LIN {X 0,Y 191.599,Z 487.439,A -85,B 0,C 180,E1 -22378.178,E2 -22378.178} C_VEL
LIN {X 0,Y 188.775,Z 497.388,A -85,B 0,C 180,E1 -22380.443,E2 -22380.443} C_VEL
LIN {X 0,Y 185.751,Z 506.671,A -85,B 0,C 180,E1 -22382.998,E2 -22382.998} C_VEL
LIN {X 0,Y 182.834,Z 515.984,A -85,B 0,C 180,E1 -22386.196,E2 -22386.196} C_VEL
LIN {X 0,Y 180.386,Z 523.716,A -85,B 0,C 180,E1 -22389.473,E2 -22389.473} C_VEL
LIN {X 0,Y 178.668,Z 530.164,A -85,B 0,C 180,E1 -22392.842,E2 -22392.842} C_VEL
LIN {X 0,Y 177.27,Z 535.423,A -85,B 0,C 180,E1 -22396.239,E2 -22396.239} C_VEL
LIN {X 0,Y 176.509,Z 539.701,A -85,B 0,C 180,E1 -22399.678,E2 -22399.678} C_VEL
LIN {X 0,Y 176.094,Z 543.09,A -85,B 0,C 180,E1 -22403.123,E2 -22403.123} C_VEL
LIN {X 0,Y 175.98,Z 546.233,A -85,B 0,C 180,E1 -22407.711,E2 -22407.711} C_VEL
LIN {X 0,Y 176.11,Z 547.274,A -85,B 0,C 180,E1 -22410,E2 -22410} C_VEL
LIN {X 0,Y 175.951,Z 548.313,A -85,B 0,C 180,E1 -22414.582,E2 -22414.582} C_VEL
LIN {X 0,Y 176.358,Z 548.034,A -85,B 0,C 180,E1 -22419.172,E2 -22419.172} C_VEL
LIN {X 0,Y 177.547,Z 546.453,A -85,B 0,C 180,E1 -22423.739,E2 -22423.739} C_VEL
LIN {X 0,Y 179.835,Z 543.544,A -85,B 0,C 180,E1 -22428.218,E2 -22428.218} C_VEL
LIN {X 0,Y 182.971,Z 539.228,A -85,B 0,C 180,E1 -22432.587,E2 -22432.587} C_VEL
LIN {X 0,Y 187.233,Z 533.386,A -85,B 0,C 180,E1 -22436.771,E2 -22436.771} C_VEL
LIN {X 0,Y 191.773,Z 526.85,A -85,B 0,C 180,E1 -22440.258,E2 -22440.258} C_VEL
LIN {X 0,Y 197.063,Z 518.782,A -85,B 0,C 180,E1 -22443.557,E2 -22443.557} C_VEL
LIN {X 0,Y 202.154,Z 510.365,A -85,B 0,C 180,E1 -22446.228,E2 -22446.228} C_VEL
LIN {X 0,Y 207.47,Z 500.385,A -85,B 0,C 180,E1 -22448.764,E2 -22448.764} C_VEL
LIN {X 0,Y 212.439,Z 490.125,A -85,B 0,C 180,E1 -22450.795,E2 -22450.795} C_VEL
LIN {X 0,Y 217.646,Z 477.789,A -85,B 0,C 180,E1 -22452.695,E2 -22452.695} C_VEL
LIN {X 0,Y 221.984,Z 465.612,A -85,B 0,C 180,E1 -22454.147,E2 -22454.147} C_VEL
LIN {X 0,Y 225.952,Z 452.09,A -85,B 0,C 180,E1 -22455.356,E2 -22455.356} C_VEL
LIN {X 0,Y 229.131,Z 437.931,A -85,B 0,C 180,E1 -22456.278,E2 -22456.278} C_VEL
LIN {X 0,Y 231.408,Z 423.369,A -85,B 0,C 180,E1 -22456.916,E2 -22456.916} C_VEL
LIN {X 0,Y 235.491,Z 369.623,A -85,B 0,C 180,E1 -22458.417,E2 -22458.417} C_VEL
LIN {X 0,Y 230.901,Z 358.639,A -85,B 0,C 180,E1 -22460.636,E2 -22460.636} C_VEL
LIN {X 0,Y 226.425,Z 349.412,A -85,B 0,C 180,E1 -22462.945,E2 -22462.945} C_VEL
LIN {X 0,Y 221.453,Z 340.153,A -85,B 0,C 180,E1 -22465.762,E2 -22465.762} C_VEL
LIN {X 0,Y 217.127,Z 332.644,A -85,B 0,C 180,E1 -22468.519,E2 -22468.519} C_VEL
LIN {X 0,Y 213.375,Z 326.679,A -85,B 0,C 180,E1 -22471.251,E2 -22471.251} C_VEL
LIN {X 0,Y 210.205,Z 321.75,A -85,B 0,C 180,E1 -22473.925,E2 -22473.925} C_VEL
LIN {X 0,Y 206.082,Z 315.639,A -85,B 0,C 180,E1 -22478.162,E2 -22478.162} C_VEL
LIN {X 0,Y 203.31,Z 313.098,A -85,B 0,C 180,E1 -22481.708,E2 -22481.708} C_VEL
LIN {X 0,Y 202.069,Z 310.201,A -85,B 0,C 180,E1 -22484.169,E2 -22484.169} C_VEL
LIN {X 0,Y 199.716,Z 308.658,A -85,B 0,C 180,E1 -22491.906,E2 -22491.906} C_VEL
LIN {X 0,Y 200.848,Z 309.272,A -85,B 0,C 180,E1 -22499.496,E2 -22499.496} C_VEL
LIN {X 0,Y 202.332,Z 310.353,A -85,B 0,C 180,E1 -22502.735,E2 -22502.735} C_VEL
LIN {X 0,Y 203.891,Z 313.395,A -85,B 0,C 180,E1 -22505.526,E2 -22505.526} C_VEL
LIN {X 0,Y 206.375,Z 315.736,A -85,B 0,C 180,E1 -22508.566,E2 -22508.566} C_VEL
LIN {X 0,Y 208.594,Z 319.275,A -85,B 0,C 180,E1 -22510.97,E2 -22510.97} C_VEL
LIN {X 0,Y 210.431,Z 321.211,A -85,B 0,C 180,E1 -22512.619,E2 -22512.619} C_VEL
LIN {X 0,Y 213.321,Z 325.119,A -85,B 0,C 180,E1 -22515.004,E2 -22515.004} C_VEL
LIN {X 0,Y 217.334,Z 330.84,A -85,B 0,C 180,E1 -22517.888,E2 -22517.888} C_VEL
LIN {X 0,Y 221.168,Z 336.313,A -85,B 0,C 180,E1 -22520.267,E2 -22520.267} C_VEL
LIN {X 0,Y 226.928,Z 345.152,A -85,B 0,C 180,E1 -22523.433,E2 -22523.433} C_VEL
LIN {X 0,Y 230.977,Z 352.505,A -85,B 0,C 180,E1 -22525.475,E2 -22525.475} C_VEL
LIN {X 0,Y 235.865,Z 362.778,A -85,B 0,C 180,E1 -22527.784,E2 -22527.784} C_VEL
LIN {X 0,Y 231.891,Z 415.14,A -85,B 0,C 180,E1 -22529.244,E2 -22529.244} C_VEL
LIN {X 0,Y 229.732,Z 429.687,A -85,B 0,C 180,E1 -22529.912,E2 -22529.912} C_VEL
LIN {X 0,Y 226.709,Z 443.815,A -85,B 0,C 180,E1 -22530.875,E2 -22530.875} C_VEL
LIN {X 0,Y 223.245,Z 456.349,A -85,B 0,C 180,E1 -22532.041,E2 -22532.041} C_VEL
LIN {X 0,Y 219.149,Z 468.478,A -85,B 0,C 180,E1 -22533.511,E2 -22533.511} C_VEL
LIN {X 0,Y 214.377,Z 480.398,A -85,B 0,C 180,E1 -22535.367,E2 -22535.367} C_VEL
LIN {X 0,Y 209.445,Z 490.898,A -85,B 0,C 180,E1 -22537.427,E2 -22537.427} C_VEL
LIN {X 0,Y 204.004,Z 501.09,A -85,B 0,C 180,E1 -22539.96,E2 -22539.96} C_VEL
LIN {X 0,Y 198.765,Z 509.97,A -85,B 0,C 180,E1 -22542.805,E2 -22542.805} C_VEL
LIN {X 0,Y 193.954,Z 517.278,A -85,B 0,C 180,E1 -22545.772,E2 -22545.772} C_VEL
LIN {X 0,Y 189.097,Z 524.169,A -85,B 0,C 180,E1 -22549.429,E2 -22549.429} C_VEL
LIN {X 0,Y 185.565,Z 528.877,A -85,B 0,C 180,E1 -22552.702,E2 -22552.702} C_VEL
LIN {X 0,Y 182.542,Z 532.562,A -85,B 0,C 180,E1 -22556.066,E2 -22556.066} C_VEL
LIN {X 0,Y 180.148,Z 535.354,A -85,B 0,C 180,E1 -22559.526,E2 -22559.526} C_VEL
LIN {X 0,Y 177.802,Z 537.718,A -85,B 0,C 180,E1 -22564.228,E2 -22564.228} C_VEL
LIN {X 0,Y 176.335,Z 538.64,A -85,B 0,C 180,E1 -22568.98,E2 -22568.98} C_VEL
LIN {X 0,Y 175.773,Z 538.153,A -85,B 0,C 180,E1 -22573.747,E2 -22573.747} C_VEL
LIN {X 0,Y 175.656,Z 536.288,A -85,B 0,C 180,E1 -22578.461,E2 -22578.461} C_VEL
LIN {X 0,Y 176.209,Z 533.006,A -85,B 0,C 180,E1 -22583.128,E2 -22583.128} C_VEL
LIN {X 0,Y 176.982,Z 529.54,A -85,B 0,C 180,E1 -22586.585,E2 -22586.585} C_VEL
LIN {X 0,Y 178.416,Z 523.586,A -85,B 0,C 180,E1 -22591.129,E2 -22591.129} C_VEL
LIN {X 0,Y 180.399,Z 516.872,A -85,B 0,C 180,E1 -22595.029,E2 -22595.029} C_VEL
LIN {X 0,Y 183.06,Z 508.512,A -85,B 0,C 180,E1 -22598.834,E2 -22598.834} C_VEL
LIN {X 0,Y 185.895,Z 499.796,A -85,B 0,C 180,E1 -22602.001,E2 -22602.001} C_VEL
LIN {X 0,Y 189.223,Z 489.232,A -85,B 0,C 180,E1 -22605.069,E2 -22605.069} C_VEL
LIN {X 0,Y 192.63,Z 477.416,A -85,B 0,C 180,E1 -22607.792,E2 -22607.792} C_VEL
LIN {X 0,Y 195.58,Z 465.587,A -85,B 0,C 180,E1 -22609.96,E2 -22609.96} C_VEL
LIN {X 0,Y 198.157,Z 454.251,A -85,B 0,C 180,E1 -22611.59,E2 -22611.59} C_VEL
LIN {X 0,Y 200.663,Z 441.026,A -85,B 0,C 180,E1 -22613.068,E2 -22613.068} C_VEL
LIN {X 0,Y 202.616,Z 426.751,A -85,B 0,C 180,E1 -22614.256,E2 -22614.256} C_VEL
LIN {X 0,Y 204.006,Z 412.463,A -85,B 0,C 180,E1 -22615.027,E2 -22615.027} C_VEL
LIN {X 0,Y 208.114,Z 340.341,A -85,B 0,C 180,E1 -22617.315,E2 -22617.315} C_VEL
LIN {X 0,Y 203.57,Z 328.395,A -85,B 0,C 180,E1 -22618.771,E2 -22618.771} C_VEL
LIN {X 0,Y 195.628,Z 313.308,A -85,B 0,C 180,E1 -22621.27,E2 -22621.27} C_VEL
LIN {X 0,Y 188.469,Z 301.599,A -85,B 0,C 180,E1 -22623.689,E2 -22623.689} C_VEL
LIN {X 0,Y 183.578,Z 294.334,A -85,B 0,C 180,E1 -22625.471,E2 -22625.471} C_VEL
LIN {X 0,Y 181.208,Z 290.635,A -85,B 0,C 180,E1 -22626.393,E2 -22626.393} C_VEL
LIN {X 0,Y 179.254,Z 288.283,A -85,B 0,C 180,E1 -22627.143,E2 -22627.143} C_VEL
LIN {X 0,Y 178.516,Z 285.874,A -85,B 0,C 180,E1 -22627.554,E2 -22627.554} C_VEL
LIN {X 0,Y 178.498,Z 285.866,A -85,B 0,C 180,E1 -22632.015,E2 -22632.015} C_VEL
LIN {X 0,Y 178.52,Z 285.859,A -85,B 0,C 180,E1 -22635.122,E2 -22635.122} C_VEL
LIN {X 0,Y 178.508,Z 285.86,A -85,B 0,C 180,E1 -22638.42,E2 -22638.42} C_VEL
LIN {X 0,Y 178.46,Z 285.851,A -85,B 0,C 180,E1 -22643.796,E2 -22643.796} C_VEL
LIN {X 0,Y 178.484,Z 285.864,A -85,B 0,C 180,E1 -22646.55,E2 -22646.55} C_VEL
LIN {X 0,Y 178.516,Z 285.865,A -85,B 0,C 180,E1 -22650.009,E2 -22650.009} C_VEL
LIN {X 0,Y 178.518,Z 285.851,A -85,B 0,C 180,E1 -22654.885,E2 -22654.885} C_VEL
LIN {X 0,Y 178.618,Z 285.853,A -85,B 0,C 180,E1 -22660.787,E2 -22660.787} C_VEL
LIN {X 0,Y 178.653,Z 285.849,A -85,B 0,C 180,E1 -22666.351,E2 -22666.351} C_VEL
LIN {X 0,Y 178.907,Z 285.804,A -85,B 0,C 180,E1 -22670.963,E2 -22670.963} C_VEL
LIN {X 0,Y 179.149,Z 285.793,A -85,B 0,C 180,E1 -22677.755,E2 -22677.755} C_VEL
LIN {X 0,Y 179.367,Z 285.757,A -85,B 0,C 180,E1 -22680.003,E2 -22680.003} C_VEL
LIN {X 0,Y 178.862,Z 285.804,A -85,B 0,C 180,E1 -22684.51,E2 -22684.51} C_VEL
LIN {X 0,Y 178.91,Z 285.821,A -85,B 0,C 180,E1 -22689.043,E2 -22689.043} C_VEL
LIN {X 0,Y 178.655,Z 285.83,A -85,B 0,C 180,E1 -22693.655,E2 -22693.655} C_VEL
LIN {X 0,Y 178.621,Z 285.852,A -85,B 0,C 180,E1 -22699.216,E2 -22699.216} C_VEL
LIN {X 0,Y 178.521,Z 285.872,A -85,B 0,C 180,E1 -22705.117,E2 -22705.117} C_VEL
LIN {X 0,Y 178.525,Z 285.871,A -85,B 0,C 180,E1 -22709.996,E2 -22709.996} C_VEL
LIN {X 0,Y 178.487,Z 285.873,A -85,B 0,C 180,E1 -22714.221,E2 -22714.221} C_VEL
LIN {X 0,Y 178.461,Z 286.066,A -85,B 0,C 180,E1 -22718.1,E2 -22718.1} C_VEL
LIN {X 0,Y 179.328,Z 288.615,A -85,B 0,C 180,E1 -22718.527,E2 -22718.527} C_VEL
LIN {X 0,Y 181.633,Z 291.388,A -85,B 0,C 180,E1 -22719.409,E2 -22719.409} C_VEL
LIN {X 0,Y 184,Z 294.886,A -85,B 0,C 180,E1 -22720.314,E2 -22720.314} C_VEL
LIN {X 0,Y 187.709,Z 300.898,A -85,B 0,C 180,E1 -22721.688,E2 -22721.688} C_VEL
LIN {X 0,Y 194.217,Z 313.493,A -85,B 0,C 180,E1 -22724.019,E2 -22724.019} C_VEL
LIN {X 0,Y 200.32,Z 326.993,A -85,B 0,C 180,E1 -22726.083,E2 -22726.083} C_VEL
LIN {X 0,Y 206.79,Z 344.301,A -85,B 0,C 180,E1 -22728.211,E2 -22728.211} C_VEL
LIN {X 0,Y 207.653,Z 350.597,A -85,B 0,C 180,E1 -22728.65,E2 -22728.65} C_VEL
LIN {X 0,Y 205.055,Z 399.727,A -85,B 0,C 180,E1 -22730.218,E2 -22730.218} C_VEL
LIN {X 0,Y 204.232,Z 405.578,A -85,B 0,C 180,E1 -22730.296,E2 -22730.296} C_VEL
LIN {X 0,Y 198.314,Z 424.511,A -85,B 0,C 180,E1 -22730.052,E2 -22730.052} C_VEL
LIN {X 0,Y 197.12,Z 430.265,A -85,B 0,C 180,E1 -22730.247,E2 -22730.247} C_VEL
LIN {X 0,Y 195.345,Z 443.358,A -85,B 0,C 180,E1 -22731.146,E2 -22731.146} C_VEL
LIN {X 0,Y 192.903,Z 456.479,A -85,B 0,C 180,E1 -22732.393,E2 -22732.393} C_VEL
LIN {X 0,Y 189.9,Z 469.458,A -85,B 0,C 180,E1 -22734.044,E2 -22734.044} C_VEL
LIN {X 0,Y 186.72,Z 482.513,A -85,B 0,C 180,E1 -22736.278,E2 -22736.278} C_VEL
LIN {X 0,Y 183.793,Z 492.107,A -85,B 0,C 180,E1 -22738.28,E2 -22738.28} C_VEL
LIN {X 0,Y 180.587,Z 502.213,A -85,B 0,C 180,E1 -22740.892,E2 -22740.892} C_VEL
LIN {X 0,Y 177.225,Z 512.26,A -85,B 0,C 180,E1 -22744.138,E2 -22744.138} C_VEL
LIN {X 0,Y 174.538,Z 520.595,A -85,B 0,C 180,E1 -22747.511,E2 -22747.511} C_VEL
LIN {X 0,Y 172.095,Z 528.543,A -85,B 0,C 180,E1 -22751.549,E2 -22751.549} C_VEL
LIN {X 0,Y 170.328,Z 534.902,A -85,B 0,C 180,E1 -22755.666,E2 -22755.666} C_VEL
LIN {X 0,Y 169.291,Z 540.513,A -85,B 0,C 180,E1 -22760.441,E2 -22760.441} C_VEL
LIN {X 0,Y 169.015,Z 542.701,A -85,B 0,C 180,E1 -22762.834,E2 -22762.834} C_VEL
LIN {X 0,Y 168.894,Z 545.923,A -85,B 0,C 180,E1 -22767.615,E2 -22767.615} C_VEL
LIN {X 0,Y 169.017,Z 546.996,A -85,B 0,C 180,E1 -22770,E2 -22770} C_VEL
LIN {X 0,Y 168.865,Z 548.097,A -85,B 0,C 180,E1 -22774.774,E2 -22774.774} C_VEL
LIN {X 0,Y 169.328,Z 547.881,A -85,B 0,C 180,E1 -22779.556,E2 -22779.556} C_VEL
LIN {X 0,Y 170.609,Z 546.362,A -85,B 0,C 180,E1 -22784.309,E2 -22784.309} C_VEL
LIN {X 0,Y 173.061,Z 543.518,A -85,B 0,C 180,E1 -22788.958,E2 -22788.958} C_VEL
LIN {X 0,Y 176.655,Z 538.932,A -85,B 0,C 180,E1 -22793.785,E2 -22793.785} C_VEL
LIN {X 0,Y 180.898,Z 533.512,A -85,B 0,C 180,E1 -22797.787,E2 -22797.787} C_VEL
LIN {X 0,Y 185.656,Z 527.059,A -85,B 0,C 180,E1 -22801.365,E2 -22801.365} C_VEL
LIN {X 0,Y 191.196,Z 519.083,A -85,B 0,C 180,E1 -22804.732,E2 -22804.732} C_VEL
LIN {X 0,Y 196.487,Z 510.766,A -85,B 0,C 180,E1 -22807.448,E2 -22807.448} C_VEL
LIN {X 0,Y 202.357,Z 500.267,A -85,B 0,C 180,E1 -22810.172,E2 -22810.172} C_VEL
LIN {X 0,Y 207.688,Z 489.714,A -85,B 0,C 180,E1 -22812.263,E2 -22812.263} C_VEL
LIN {X 0,Y 213.051,Z 477.329,A -85,B 0,C 180,E1 -22814.174,E2 -22814.174} C_VEL
LIN {X 0,Y 217.574,Z 465.082,A -85,B 0,C 180,E1 -22815.615,E2 -22815.615} C_VEL
LIN {X 0,Y 221.628,Z 451.483,A -85,B 0,C 180,E1 -22816.83,E2 -22816.83} C_VEL
LIN {X 0,Y 224.944,Z 437.181,A -85,B 0,C 180,E1 -22817.736,E2 -22817.736} C_VEL
LIN {X 0,Y 227.194,Z 423.145,A -85,B 0,C 180,E1 -22818.339,E2 -22818.339} C_VEL
LIN {X 0,Y 231.149,Z 372.075,A -85,B 0,C 180,E1 -22819.801,E2 -22819.801} C_VEL
LIN {X 0,Y 226.57,Z 361.295,A -85,B 0,C 180,E1 -22822.17,E2 -22822.17} C_VEL
LIN {X 0,Y 222.235,Z 352.184,A -85,B 0,C 180,E1 -22824.597,E2 -22824.597} C_VEL
LIN {X 0,Y 217.151,Z 342.693,A -85,B 0,C 180,E1 -22827.752,E2 -22827.752} C_VEL
LIN {X 0,Y 212.407,Z 334.425,A -85,B 0,C 180,E1 -22831.201,E2 -22831.201} C_VEL
LIN {X 0,Y 208.423,Z 328.16,A -85,B 0,C 180,E1 -22834.648,E2 -22834.648} C_VEL
LIN {X 0,Y 204.763,Z 322.459,A -85,B 0,C 180,E1 -22838.61,E2 -22838.61} C_VEL
LIN {X 0,Y 202.118,Z 319.903,A -85,B 0,C 180,E1 -22842.17,E2 -22842.17} C_VEL
LIN {X 0,Y 200.885,Z 317.174,A -85,B 0,C 180,E1 -22844.729,E2 -22844.729} C_VEL
LIN {X 0,Y 198.844,Z 315.713,A -85,B 0,C 180,E1 -22851.87,E2 -22851.87} C_VEL
LIN {X 0,Y 199.968,Z 316.325,A -85,B 0,C 180,E1 -22859.494,E2 -22859.494} C_VEL
LIN {X 0,Y 201.222,Z 317.276,A -85,B 0,C 180,E1 -22862.327,E2 -22862.327} C_VEL
LIN {X 0,Y 202.8,Z 320.36,A -85,B 0,C 180,E1 -22865.263,E2 -22865.263} C_VEL
LIN {X 0,Y 205.027,Z 322.627,A -85,B 0,C 180,E1 -22868.113,E2 -22868.113} C_VEL
LIN {X 0,Y 207.417,Z 326.287,A -85,B 0,C 180,E1 -22870.755,E2 -22870.755} C_VEL
LIN {X 0,Y 208.836,Z 327.902,A -85,B 0,C 180,E1 -22872.077,E2 -22872.077} C_VEL
LIN {X 0,Y 212.21,Z 332.715,A -85,B 0,C 180,E1 -22874.946,E2 -22874.946} C_VEL
LIN {X 0,Y 215.576,Z 337.605,A -85,B 0,C 180,E1 -22877.426,E2 -22877.426} C_VEL
LIN {X 0,Y 220.029,Z 344.131,A -85,B 0,C 180,E1 -22880.249,E2 -22880.249} C_VEL
LIN {X 0,Y 225.73,Z 353.527,A -85,B 0,C 180,E1 -22883.442,E2 -22883.442} C_VEL
LIN {X 0,Y 230.588,Z 363.521,A -85,B 0,C 180,E1 -22885.947,E2 -22885.947} C_VEL
LIN {X 0,Y 231.586,Z 365.841,A -85,B 0,C 180,E1 -22886.443,E2 -22886.443} C_VEL
LIN {X 0,Y 227.745,Z 414.733,A -85,B 0,C 180,E1 -22887.804,E2 -22887.804} C_VEL
LIN {X 0,Y 225.513,Z 429.496,A -85,B 0,C 180,E1 -22888.471,E2 -22888.471} C_VEL
LIN {X 0,Y 222.393,Z 443.676,A -85,B 0,C 180,E1 -22889.425,E2 -22889.425} C_VEL
LIN {X 0,Y 218.866,Z 456.059,A -85,B 0,C 180,E1 -22890.563,E2 -22890.563} C_VEL
LIN {X 0,Y 214.572,Z 468.45,A -85,B 0,C 180,E1 -22892.062,E2 -22892.062} C_VEL
LIN {X 0,Y 209.611,Z 480.408,A -85,B 0,C 180,E1 -22893.92,E2 -22893.92} C_VEL
LIN {X 0,Y 203.966,Z 491.947,A -85,B 0,C 180,E1 -22896.209,E2 -22896.209} C_VEL
LIN {X 0,Y 198.318,Z 501.969,A -85,B 0,C 180,E1 -22898.775,E2 -22898.775} C_VEL
LIN {X 0,Y 192.874,Z 510.714,A -85,B 0,C 180,E1 -22901.672,E2 -22901.672} C_VEL
LIN {X 0,Y 187.85,Z 517.932,A -85,B 0,C 180,E1 -22904.698,E2 -22904.698} C_VEL
LIN {X 0,Y 183.465,Z 523.866,A -85,B 0,C 180,E1 -22907.906,E2 -22907.906} C_VEL
LIN {X 0,Y 179.213,Z 529.174,A -85,B 0,C 180,E1 -22911.652,E2 -22911.652} C_VEL
LIN {X 0,Y 175.409,Z 533.532,A -85,B 0,C 180,E1 -22915.881,E2 -22915.881} C_VEL
LIN {X 0,Y 172.262,Z 536.754,A -85,B 0,C 180,E1 -22920.688,E2 -22920.688} C_VEL
LIN {X 0,Y 170.184,Z 538.489,A -85,B 0,C 180,E1 -22925.61,E2 -22925.61} C_VEL
LIN {X 0,Y 168.945,Z 538.803,A -85,B 0,C 180,E1 -22930.562,E2 -22930.562} C_VEL
LIN {X 0,Y 168.674,Z 538.361,A -85,B 0,C 180,E1 -22933.387,E2 -22933.387} C_VEL
LIN {X 0,Y 168.53,Z 536.661,A -85,B 0,C 180,E1 -22937.966,E2 -22937.966} C_VEL
LIN {X 0,Y 169.046,Z 533.488,A -85,B 0,C 180,E1 -22942.836,E2 -22942.836} C_VEL
LIN {X 0,Y 169.829,Z 530.109,A -85,B 0,C 180,E1 -22946.441,E2 -22946.441} C_VEL
LIN {X 0,Y 171.302,Z 524.262,A -85,B 0,C 180,E1 -22951.176,E2 -22951.176} C_VEL
LIN {X 0,Y 173.302,Z 517.678,A -85,B 0,C 180,E1 -22955.235,E2 -22955.235} C_VEL
LIN {X 0,Y 176.021,Z 509.508,A -85,B 0,C 180,E1 -22959.19,E2 -22959.19} C_VEL
LIN {X 0,Y 178.96,Z 500.948,A -85,B 0,C 180,E1 -22962.474,E2 -22962.474} C_VEL
LIN {X 0,Y 182.367,Z 490.582,A -85,B 0,C 180,E1 -22965.65,E2 -22965.65} C_VEL
LIN {X 0,Y 185.915,Z 478.99,A -85,B 0,C 180,E1 -22968.457,E2 -22968.457} C_VEL
LIN {X 0,Y 188.984,Z 467.448,A -85,B 0,C 180,E1 -22970.688,E2 -22970.688} C_VEL
LIN {X 0,Y 191.538,Z 456.54,A -85,B 0,C 180,E1 -22972.376,E2 -22972.376} C_VEL
LIN {X 0,Y 194.173,Z 443.872,A -85,B 0,C 180,E1 -22973.886,E2 -22973.886} C_VEL
LIN {X 0,Y 196.319,Z 429.762,A -85,B 0,C 180,E1 -22975.157,E2 -22975.157} C_VEL
LIN {X 0,Y 197.909,Z 415.615,A -85,B 0,C 180,E1 -22976.013,E2 -22976.013} C_VEL
LIN {X 0,Y 199.359,Z 392.322,A -85,B 0,C 180,E1 -22976.843,E2 -22976.843} C_VEL
LIN {X 0,Y 202.207,Z 341.799,A -85,B 0,C 180,E1 -22978.472,E2 -22978.472} C_VEL
LIN {X 0,Y 198.36,Z 331.838,A -85,B 0,C 180,E1 -22979.766,E2 -22979.766} C_VEL
LIN {X 0,Y 191.132,Z 317.879,A -85,B 0,C 180,E1 -22982.17,E2 -22982.17} C_VEL
LIN {X 0,Y 184.087,Z 306.206,A -85,B 0,C 180,E1 -22984.686,E2 -22984.686} C_VEL
LIN {X 0,Y 178.777,Z 298.299,A -85,B 0,C 180,E1 -22986.731,E2 -22986.731} C_VEL
LIN {X 0,Y 177.03,Z 295.69,A -85,B 0,C 180,E1 -22987.446,E2 -22987.446} C_VEL
LIN {X 0,Y 174.901,Z 292.466,A -85,B 0,C 180,E1 -22988.353,E2 -22988.353} C_VEL
LIN {X 0,Y 174.113,Z 291.47,A -85,B 0,C 180,E1 -22988.686,E2 -22988.686} C_VEL
LIN {X 0,Y 172.088,Z 289.03,A -85,B 0,C 180,E1 -22989.559,E2 -22989.559} C_VEL
LIN {X 0,Y 171.411,Z 286.741,A -85,B 0,C 180,E1 -22990.023,E2 -22990.023} C_VEL
LIN {X 0,Y 171.442,Z 286.751,A -85,B 0,C 180,E1 -22994.177,E2 -22994.177} C_VEL
LIN {X 0,Y 171.425,Z 286.748,A -85,B 0,C 180,E1 -22999.012,E2 -22999.012} C_VEL
LIN {X 0,Y 171.434,Z 286.74,A -85,B 0,C 180,E1 -23002.058,E2 -23002.058} C_VEL
LIN {X 0,Y 171.421,Z 286.754,A -85,B 0,C 180,E1 -23007.797,E2 -23007.797} C_VEL
LIN {X 0,Y 171.442,Z 286.739,A -85,B 0,C 180,E1 -23010.537,E2 -23010.537} C_VEL
LIN {X 0,Y 171.447,Z 286.74,A -85,B 0,C 180,E1 -23015.804,E2 -23015.804} C_VEL
LIN {X 0,Y 171.574,Z 286.73,A -85,B 0,C 180,E1 -23020.875,E2 -23020.875} C_VEL
LIN {X 0,Y 171.571,Z 286.729,A -85,B 0,C 180,E1 -23025.776,E2 -23025.776} C_VEL
LIN {X 0,Y 171.844,Z 286.687,A -85,B 0,C 180,E1 -23030.588,E2 -23030.588} C_VEL
LIN {X 0,Y 171.811,Z 286.688,A -85,B 0,C 180,E1 -23035.311,E2 -23035.311} C_VEL
LIN {X 0,Y 172.329,Z 286.633,A -85,B 0,C 180,E1 -23040.003,E2 -23040.003} C_VEL
LIN {X 0,Y 171.811,Z 286.683,A -85,B 0,C 180,E1 -23044.696,E2 -23044.696} C_VEL
LIN {X 0,Y 171.847,Z 286.697,A -85,B 0,C 180,E1 -23049.418,E2 -23049.418} C_VEL
LIN {X 0,Y 171.573,Z 286.716,A -85,B 0,C 180,E1 -23054.231,E2 -23054.231} C_VEL
LIN {X 0,Y 171.54,Z 286.734,A -85,B 0,C 180,E1 -23059.56,E2 -23059.56} C_VEL
LIN {X 0,Y 171.46,Z 286.753,A -85,B 0,C 180,E1 -23065.612,E2 -23065.612} C_VEL
LIN {X 0,Y 171.443,Z 286.75,A -85,B 0,C 180,E1 -23070.589,E2 -23070.589} C_VEL
LIN {X 0,Y 171.393,Z 286.814,A -85,B 0,C 180,E1 -23075.668,E2 -23075.668} C_VEL
LIN {X 0,Y 172.308,Z 289.471,A -85,B 0,C 180,E1 -23076.17,E2 -23076.17} C_VEL
LIN {X 0,Y 174.335,Z 291.706,A -85,B 0,C 180,E1 -23077.029,E2 -23077.029} C_VEL
LIN {X 0,Y 176.961,Z 295.713,A -85,B 0,C 180,E1 -23078.158,E2 -23078.158} C_VEL
LIN {X 0,Y 178.596,Z 298.091,A -85,B 0,C 180,E1 -23078.827,E2 -23078.827} C_VEL
LIN {X 0,Y 182.642,Z 304.082,A -85,B 0,C 180,E1 -23080.405,E2 -23080.405} C_VEL
LIN {X 0,Y 189.835,Z 318.338,A -85,B 0,C 180,E1 -23083.14,E2 -23083.14} C_VEL
LIN {X 0,Y 195.529,Z 331.21,A -85,B 0,C 180,E1 -23085.176,E2 -23085.176} C_VEL
LIN {X 0,Y 201.519,Z 347.777,A -85,B 0,C 180,E1 -23087.273,E2 -23087.273} C_VEL
LIN {X 0,Y 201.822,Z 352.981,A -85,B 0,C 180,E1 -23087.566,E2 -23087.566} C_VEL
LIN {X 0,Y 197.799,Z 423.508,A -85,B 0,C 180,E1 -23089.906,E2 -23089.906} C_VEL
LIN {X 0,Y 197.12,Z 430.265,A -85,B 0,C 180,E1 -23090.247,E2 -23090.247} C_VEL
LIN {X 0,Y 196.033,Z 434.097,A -85,B 0,C 180,E1 -23090.355,E2 -23090.355} C_VEL
LIN {X 0,Y 189.413,Z 445.895,A -85,B 0,C 180,E1 -23090.283,E2 -23090.283} C_VEL
LIN {X 0,Y 188.223,Z 449.593,A -85,B 0,C 180,E1 -23090.533,E2 -23090.533} C_VEL
LIN {X 0,Y 185.525,Z 462.569,A -85,B 0,C 180,E1 -23092.007,E2 -23092.007} C_VEL
LIN {X 0,Y 182.835,Z 473.325,A -85,B 0,C 180,E1 -23093.568,E2 -23093.568} C_VEL
LIN {X 0,Y 179.691,Z 485.184,A -85,B 0,C 180,E1 -23095.79,E2 -23095.79} C_VEL
LIN {X 0,Y 177.365,Z 492.134,A -85,B 0,C 180,E1 -23097.325,E2 -23097.325} C_VEL
LIN {X 0,Y 174.359,Z 501.302,A -85,B 0,C 180,E1 -23099.746,E2 -23099.746} C_VEL
LIN {X 0,Y 170.81,Z 511.469,A -85,B 0,C 180,E1 -23103.09,E2 -23103.09} C_VEL
LIN {X 0,Y 167.941,Z 519.902,A -85,B 0,C 180,E1 -23106.575,E2 -23106.575} C_VEL
LIN {X 0,Y 165.681,Z 526.92,A -85,B 0,C 180,E1 -23110.163,E2 -23110.163} C_VEL
LIN {X 0,Y 163.914,Z 532.727,A -85,B 0,C 180,E1 -23113.818,E2 -23113.818} C_VEL
LIN {X 0,Y 162.699,Z 537.434,A -85,B 0,C 180,E1 -23117.527,E2 -23117.527} C_VEL
LIN {X 0,Y 162.105,Z 541.219,A -85,B 0,C 180,E1 -23121.272,E2 -23121.272} C_VEL
LIN {X 0,Y 161.801,Z 544.136,A -85,B 0,C 180,E1 -23125.016,E2 -23125.016} C_VEL
LIN {X 0,Y 161.927,Z 546.716,A -85,B 0,C 180,E1 -23130,E2 -23130} C_VEL
LIN {X 0,Y 161.804,Z 547.466,A -85,B 0,C 180,E1 -23132.489,E2 -23132.489} C_VEL
LIN {X 0,Y 161.937,Z 547.967,A -85,B 0,C 180,E1 -23137.481,E2 -23137.481} C_VEL
LIN {X 0,Y 162.876,Z 547.163,A -85,B 0,C 180,E1 -23142.459,E2 -23142.459} C_VEL
LIN {X 0,Y 164.878,Z 545.055,A -85,B 0,C 180,E1 -23147.36,E2 -23147.36} C_VEL
LIN {X 0,Y 167.986,Z 541.594,A -85,B 0,C 180,E1 -23152.118,E2 -23152.118} C_VEL
LIN {X 0,Y 172.103,Z 536.682,A -85,B 0,C 180,E1 -23156.691,E2 -23156.691} C_VEL
LIN {X 0,Y 177.403,Z 530.176,A -85,B 0,C 180,E1 -23160.997,E2 -23160.997} C_VEL
LIN {X 0,Y 182.803,Z 522.975,A -85,B 0,C 180,E1 -23164.545,E2 -23164.545} C_VEL
LIN {X 0,Y 189.043,Z 514.105,A -85,B 0,C 180,E1 -23167.836,E2 -23167.836} C_VEL
LIN {X 0,Y 194.748,Z 504.847,A -85,B 0,C 180,E1 -23170.508,E2 -23170.508} C_VEL
LIN {X 0,Y 200.333,Z 494.655,A -85,B 0,C 180,E1 -23172.819,E2 -23172.819} C_VEL
LIN {X 0,Y 205.854,Z 483.44,A -85,B 0,C 180,E1 -23174.759,E2 -23174.759} C_VEL
LIN {X 0,Y 210.929,Z 471.105,A -85,B 0,C 180,E1 -23176.442,E2 -23176.442} C_VEL
LIN {X 0,Y 215.136,Z 459.206,A -85,B 0,C 180,E1 -23177.654,E2 -23177.654} C_VEL
LIN {X 0,Y 218.765,Z 446.242,A -85,B 0,C 180,E1 -23178.67,E2 -23178.67} C_VEL
LIN {X 0,Y 221.684,Z 432.344,A -85,B 0,C 180,E1 -23179.451,E2 -23179.451} C_VEL
LIN {X 0,Y 223.65,Z 417.686,A -85,B 0,C 180,E1 -23180.007,E2 -23180.007} C_VEL
LIN {X 0,Y 226.984,Z 374.911,A -85,B 0,C 180,E1 -23181.207,E2 -23181.207} C_VEL
LIN {X 0,Y 223.064,Z 365.487,A -85,B 0,C 180,E1 -23183.38,E2 -23183.38} C_VEL
LIN {X 0,Y 219.422,Z 357.561,A -85,B 0,C 180,E1 -23185.552,E2 -23185.552} C_VEL
LIN {X 0,Y 214.653,Z 348.38,A -85,B 0,C 180,E1 -23188.686,E2 -23188.686} C_VEL
LIN {X 0,Y 210.267,Z 340.346,A -85,B 0,C 180,E1 -23192.097,E2 -23192.097} C_VEL
LIN {X 0,Y 206.633,Z 334.465,A -85,B 0,C 180,E1 -23195.43,E2 -23195.43} C_VEL
LIN {X 0,Y 203.338,Z 329.247,A -85,B 0,C 180,E1 -23199.191,E2 -23199.191} C_VEL
LIN {X 0,Y 200.776,Z 326.405,A -85,B 0,C 180,E1 -23202.938,E2 -23202.938} C_VEL
LIN {X 0,Y 199.898,Z 324.18,A -85,B 0,C 180,E1 -23204.927,E2 -23204.927} C_VEL
LIN {X 0,Y 197.97,Z 322.761,A -85,B 0,C 180,E1 -23211.834,E2 -23211.834} C_VEL
LIN {X 0,Y 199.082,Z 323.383,A -85,B 0,C 180,E1 -23219.492,E2 -23219.492} C_VEL
LIN {X 0,Y 200.101,Z 324.14,A -85,B 0,C 180,E1 -23221.872,E2 -23221.872} C_VEL
LIN {X 0,Y 201.658,Z 327.257,A -85,B 0,C 180,E1 -23224.915,E2 -23224.915} C_VEL
LIN {X 0,Y 203.684,Z 329.475,A -85,B 0,C 180,E1 -23227.639,E2 -23227.639} C_VEL
LIN {X 0,Y 206.374,Z 333.468,A -85,B 0,C 180,E1 -23230.668,E2 -23230.668} C_VEL
LIN {X 0,Y 207.46,Z 334.939,A -85,B 0,C 180,E1 -23231.725,E2 -23231.725} C_VEL
LIN {X 0,Y 210.475,Z 339.308,A -85,B 0,C 180,E1 -23234.377,E2 -23234.377} C_VEL
LIN {X 0,Y 213.704,Z 344.18,A -85,B 0,C 180,E1 -23236.856,E2 -23236.856} C_VEL
LIN {X 0,Y 217.593,Z 350.062,A -85,B 0,C 180,E1 -23239.445,E2 -23239.445} C_VEL
LIN {X 0,Y 222.928,Z 359.153,A -85,B 0,C 180,E1 -23242.589,E2 -23242.589} C_VEL
LIN {X 0,Y 227.401,Z 368.697,A -85,B 0,C 180,E1 -23245.023,E2 -23245.023} C_VEL
LIN {X 0,Y 223.648,Z 415.206,A -85,B 0,C 180,E1 -23246.341,E2 -23246.341} C_VEL
LIN {X 0,Y 221.344,Z 429.92,A -85,B 0,C 180,E1 -23247.009,E2 -23247.009} C_VEL
LIN {X 0,Y 218.219,Z 443.605,A -85,B 0,C 180,E1 -23247.916,E2 -23247.916} C_VEL
LIN {X 0,Y 214.472,Z 456.382,A -85,B 0,C 180,E1 -23249.088,E2 -23249.088} C_VEL
LIN {X 0,Y 210.131,Z 468.471,A -85,B 0,C 180,E1 -23250.548,E2 -23250.548} C_VEL
LIN {X 0,Y 204.997,Z 480.451,A -85,B 0,C 180,E1 -23252.413,E2 -23252.413} C_VEL
LIN {X 0,Y 199.325,Z 491.639,A -85,B 0,C 180,E1 -23254.63,E2 -23254.63} C_VEL
LIN {X 0,Y 193.757,Z 501.229,A -85,B 0,C 180,E1 -23257.064,E2 -23257.064} C_VEL
LIN {X 0,Y 187.959,Z 510.154,A -85,B 0,C 180,E1 -23259.96,E2 -23259.96} C_VEL
LIN {X 0,Y 182.679,Z 517.498,A -85,B 0,C 180,E1 -23263.034,E2 -23263.034} C_VEL
LIN {X 0,Y 177.952,Z 523.523,A -85,B 0,C 180,E1 -23266.281,E2 -23266.281} C_VEL
LIN {X 0,Y 172.878,Z 529.521,A -85,B 0,C 180,E1 -23270.564,E2 -23270.564} C_VEL
LIN {X 0,Y 169.236,Z 533.421,A -85,B 0,C 180,E1 -23274.453,E2 -23274.453} C_VEL
LIN {X 0,Y 165.788,Z 536.791,A -85,B 0,C 180,E1 -23279.424,E2 -23279.424} C_VEL
LIN {X 0,Y 163.406,Z 538.632,A -85,B 0,C 180,E1 -23284.572,E2 -23284.572} C_VEL
LIN {X 0,Y 161.977,Z 539.035,A -85,B 0,C 180,E1 -23289.69,E2 -23289.69} C_VEL
LIN {X 0,Y 161.631,Z 538.558,A -85,B 0,C 180,E1 -23293.043,E2 -23293.043} C_VEL
LIN {X 0,Y 161.419,Z 537.035,A -85,B 0,C 180,E1 -23297.427,E2 -23297.427} C_VEL
LIN {X 0,Y 161.888,Z 533.958,A -85,B 0,C 180,E1 -23302.517,E2 -23302.517} C_VEL
LIN {X 0,Y 162.679,Z 530.678,A -85,B 0,C 180,E1 -23306.285,E2 -23306.285} C_VEL
LIN {X 0,Y 164.19,Z 524.938,A -85,B 0,C 180,E1 -23311.227,E2 -23311.227} C_VEL
LIN {X 0,Y 166.184,Z 518.475,A -85,B 0,C 180,E1 -23315.46,E2 -23315.46} C_VEL
LIN {X 0,Y 169.004,Z 510.443,A -85,B 0,C 180,E1 -23319.575,E2 -23319.575} C_VEL
LIN {X 0,Y 172.018,Z 502.033,A -85,B 0,C 180,E1 -23322.986,E2 -23322.986} C_VEL
LIN {X 0,Y 175.545,Z 491.904,A -85,B 0,C 180,E1 -23326.275,E2 -23326.275} C_VEL
LIN {X 0,Y 179.23,Z 480.549,A -85,B 0,C 180,E1 -23329.172,E2 -23329.172} C_VEL
LIN {X 0,Y 182.428,Z 469.285,A -85,B 0,C 180,E1 -23331.468,E2 -23331.468} C_VEL
LIN {X 0,Y 184.972,Z 458.774,A -85,B 0,C 180,E1 -23333.216,E2 -23333.216} C_VEL
LIN {X 0,Y 187.77,Z 446.619,A -85,B 0,C 180,E1 -23334.754,E2 -23334.754} C_VEL
LIN {X 0,Y 190.066,Z 432.694,A -85,B 0,C 180,E1 -23336.12,E2 -23336.12} C_VEL
LIN {X 0,Y 191.822,Z 418.327,A -85,B 0,C 180,E1 -23337.081,E2 -23337.081} C_VEL
LIN {X 0,Y 193.142,Z 399.928,A -85,B 0,C 180,E1 -23337.809,E2 -23337.809} C_VEL
LIN {X 0,Y 196.442,Z 343.511,A -85,B 0,C 180,E1 -23339.667,E2 -23339.667} C_VEL
LIN {X 0,Y 193.301,Z 335.429,A -85,B 0,C 180,E1 -23340.783,E2 -23340.783} C_VEL
LIN {X 0,Y 186.27,Z 321.653,A -85,B 0,C 180,E1 -23343.267,E2 -23343.267} C_VEL
LIN {X 0,Y 178.708,Z 309.051,A -85,B 0,C 180,E1 -23346.149,E2 -23346.149} C_VEL
LIN {X 0,Y 172.941,Z 300.564,A -85,B 0,C 180,E1 -23348.55,E2 -23348.55} C_VEL
LIN {X 0,Y 170.39,Z 296.894,A -85,B 0,C 180,E1 -23349.696,E2 -23349.696} C_VEL
LIN {X 0,Y 168.139,Z 293.746,A -85,B 0,C 180,E1 -23350.752,E2 -23350.752} C_VEL
LIN {X 0,Y 167.402,Z 292.599,A -85,B 0,C 180,E1 -23351.117,E2 -23351.117} C_VEL
LIN {X 0,Y 165.4,Z 290.497,A -85,B 0,C 180,E1 -23352.069,E2 -23352.069} C_VEL
LIN {X 0,Y 164.389,Z 287.63,A -85,B 0,C 180,E1 -23352.696,E2 -23352.696} C_VEL
LIN {X 0,Y 164.386,Z 287.608,A -85,B 0,C 180,E1 -23356.845,E2 -23356.845} C_VEL
LIN {X 0,Y 164.369,Z 287.633,A -85,B 0,C 180,E1 -23360.32,E2 -23360.32} C_VEL
LIN {X 0,Y 164.34,Z 287.606,A -85,B 0,C 180,E1 -23364.343,E2 -23364.343} C_VEL
LIN {X 0,Y 164.398,Z 287.628,A -85,B 0,C 180,E1 -23369.141,E2 -23369.141} C_VEL
LIN {X 0,Y 164.404,Z 287.603,A -85,B 0,C 180,E1 -23374.696,E2 -23374.696} C_VEL
LIN {X 0,Y 164.479,Z 287.614,A -85,B 0,C 180,E1 -23380.054,E2 -23380.054} C_VEL
LIN {X 0,Y 164.501,Z 287.61,A -85,B 0,C 180,E1 -23385.151,E2 -23385.151} C_VEL
LIN {X 0,Y 164.764,Z 287.572,A -85,B 0,C 180,E1 -23390.18,E2 -23390.18} C_VEL
LIN {X 0,Y 164.827,Z 287.541,A -85,B 0,C 180,E1 -23392.654,E2 -23392.654} C_VEL
LIN {X 0,Y 165.044,Z 287.55,A -85,B 0,C 180,E1 -23397.563,E2 -23397.563} C_VEL
LIN {X 0,Y 165.292,Z 287.509,A -85,B 0,C 180,E1 -23400.003,E2 -23400.003} C_VEL
LIN {X 0,Y 164.759,Z 287.562,A -85,B 0,C 180,E1 -23404.897,E2 -23404.897} C_VEL
LIN {X 0,Y 164.829,Z 287.578,A -85,B 0,C 180,E1 -23407.352,E2 -23407.352} C_VEL
LIN {X 0,Y 164.702,Z 287.567,A -85,B 0,C 180,E1 -23411.064,E2 -23411.064} C_VEL
LIN {X 0,Y 164.482,Z 287.622,A -85,B 0,C 180,E1 -23417.406,E2 -23417.406} C_VEL
LIN {X 0,Y 164.474,Z 287.616,A -85,B 0,C 180,E1 -23419.992,E2 -23419.992} C_VEL
LIN {X 0,Y 164.388,Z 287.632,A -85,B 0,C 180,E1 -23426.131,E2 -23426.131} C_VEL
LIN {X 0,Y 164.381,Z 287.633,A -85,B 0,C 180,E1 -23432.377,E2 -23432.377} C_VEL
LIN {X 0,Y 164.337,Z 287.641,A -85,B 0,C 180,E1 -23432.906,E2 -23432.906} C_VEL
LIN {X 0,Y 165.25,Z 290.365,A -85,B 0,C 180,E1 -23433.481,E2 -23433.481} C_VEL
LIN {X 0,Y 167.246,Z 292.53,A -85,B 0,C 180,E1 -23434.436,E2 -23434.436} C_VEL
LIN {X 0,Y 167.907,Z 293.297,A -85,B 0,C 180,E1 -23434.747,E2 -23434.747} C_VEL
LIN {X 0,Y 170.099,Z 296.641,A -85,B 0,C 180,E1 -23435.799,E2 -23435.799} C_VEL
LIN {X 0,Y 171.406,Z 298.414,A -85,B 0,C 180,E1 -23436.391,E2 -23436.391} C_VEL
LIN {X 0,Y 176.879,Z 306.338,A -85,B 0,C 180,E1 -23438.741,E2 -23438.741} C_VEL
LIN {X 0,Y 180.372,Z 312.545,A -85,B 0,C 180,E1 -23440.183,E2 -23440.183} C_VEL
LIN {X 0,Y 186.76,Z 325.894,A -85,B 0,C 180,E1 -23442.704,E2 -23442.704} C_VEL
LIN {X 0,Y 192.113,Z 339.01,A -85,B 0,C 180,E1 -23444.725,E2 -23444.725} C_VEL
LIN {X 0,Y 196.031,Z 350.366,A -85,B 0,C 180,E1 -23446.182,E2 -23446.182} C_VEL
LIN {X 0,Y 196.047,Z 355.298,A -85,B 0,C 180,E1 -23446.412,E2 -23446.412} C_VEL
LIN {X 0,Y 192.065,Z 422.729,A -85,B 0,C 180,E1 -23448.686,E2 -23448.686} C_VEL
LIN {X 0,Y 190.422,Z 437.008,A -85,B 0,C 180,E1 -23449.509,E2 -23449.509} C_VEL
LIN {X 0,Y 188.223,Z 449.593,A -85,B 0,C 180,E1 -23450.533,E2 -23450.533} C_VEL
LIN {X 0,Y 187.276,Z 453.306,A -85,B 0,C 180,E1 -23450.87,E2 -23450.87} C_VEL
LIN {X 0,Y 184.105,Z 460.43,A -85,B 0,C 180,E1 -23451.365,E2 -23451.365} C_VEL
LIN {X 0,Y 177.514,Z 472.256,A -85,B 0,C 180,E1 -23452.356,E2 -23452.356} C_VEL
LIN {X 0,Y 175.627,Z 477.217,A -85,B 0,C 180,E1 -23453.122,E2 -23453.122} C_VEL
LIN {X 0,Y 172.924,Z 486.512,A -85,B 0,C 180,E1 -23455.003,E2 -23455.003} C_VEL
LIN {X 0,Y 170.325,Z 494.319,A -85,B 0,C 180,E1 -23456.858,E2 -23456.858} C_VEL
LIN {X 0,Y 166.844,Z 503.981,A -85,B 0,C 180,E1 -23459.637,E2 -23459.637} C_VEL
LIN {X 0,Y 163.326,Z 513.678,A -85,B 0,C 180,E1 -23463.14,E2 -23463.14} C_VEL
LIN {X 0,Y 160.221,Z 522.345,A -85,B 0,C 180,E1 -23467.102,E2 -23467.102} C_VEL
LIN {X 0,Y 158.212,Z 528.355,A -85,B 0,C 180,E1 -23470.539,E2 -23470.539} C_VEL
LIN {X 0,Y 156.504,Z 533.854,A -85,B 0,C 180,E1 -23474.369,E2 -23474.369} C_VEL
LIN {X 0,Y 155.207,Z 539.615,A -85,B 0,C 180,E1 -23479.565,E2 -23479.565} C_VEL
LIN {X 0,Y 154.908,Z 541.881,A -85,B 0,C 180,E1 -23482.177,E2 -23482.177} C_VEL
LIN {X 0,Y 154.705,Z 545.267,A -85,B 0,C 180,E1 -23487.396,E2 -23487.396} C_VEL
LIN {X 0,Y 154.827,Z 546.418,A -85,B 0,C 180,E1 -23490,E2 -23490} C_VEL
LIN {X 0,Y 154.696,Z 547.657,A -85,B 0,C 180,E1 -23495.213,E2 -23495.213} C_VEL
LIN {X 0,Y 155.286,Z 547.573,A -85,B 0,C 180,E1 -23500.429,E2 -23500.429} C_VEL
LIN {X 0,Y 156.799,Z 546.187,A -85,B 0,C 180,E1 -23505.6,E2 -23505.6} C_VEL
LIN {X 0,Y 159.596,Z 543.48,A -85,B 0,C 180,E1 -23510.627,E2 -23510.627} C_VEL
LIN {X 0,Y 163.398,Z 539.38,A -85,B 0,C 180,E1 -23515.474,E2 -23515.474} C_VEL
LIN {X 0,Y 168.417,Z 533.767,A -85,B 0,C 180,E1 -23520.049,E2 -23520.049} C_VEL
LIN {X 0,Y 174.518,Z 526.474,A -85,B 0,C 180,E1 -23524.317,E2 -23524.317} C_VEL
LIN {X 0,Y 179.699,Z 519.694,A -85,B 0,C 180,E1 -23527.314,E2 -23527.314} C_VEL
LIN {X 0,Y 185.455,Z 511.592,A -85,B 0,C 180,E1 -23530.107,E2 -23530.107} C_VEL
LIN {X 0,Y 191.28,Z 502.173,A -85,B 0,C 180,E1 -23532.703,E2 -23532.703} C_VEL
LIN {X 0,Y 196.901,Z 492.181,A -85,B 0,C 180,E1 -23534.823,E2 -23534.823} C_VEL
LIN {X 0,Y 202.651,Z 480.498,A -85,B 0,C 180,E1 -23536.741,E2 -23536.741} C_VEL
LIN {X 0,Y 207.348,Z 469.112,A -85,B 0,C 180,E1 -23538.216,E2 -23538.216} C_VEL
LIN {X 0,Y 211.708,Z 456.752,A -85,B 0,C 180,E1 -23539.407,E2 -23539.407} C_VEL
LIN {X 0,Y 215.433,Z 443.112,A -85,B 0,C 180,E1 -23540.416,E2 -23540.416} C_VEL
LIN {X 0,Y 218.34,Z 428.761,A -85,B 0,C 180,E1 -23541.143,E2 -23541.143} C_VEL
LIN {X 0,Y 220.044,Z 414.846,A -85,B 0,C 180,E1 -23541.616,E2 -23541.616} C_VEL
LIN {X 0,Y 222.992,Z 377.875,A -85,B 0,C 180,E1 -23542.644,E2 -23542.644} C_VEL
LIN {X 0,Y 219.22,Z 368.572,A -85,B 0,C 180,E1 -23544.906,E2 -23544.906} C_VEL
LIN {X 0,Y 214.738,Z 358.951,A -85,B 0,C 180,E1 -23547.834,E2 -23547.834} C_VEL
LIN {X 0,Y 211.343,Z 352.334,A -85,B 0,C 180,E1 -23550.334,E2 -23550.334} C_VEL
LIN {X 0,Y 207.792,Z 345.701,A -85,B 0,C 180,E1 -23553.351,E2 -23553.351} C_VEL
LIN {X 0,Y 204.923,Z 340.855,A -85,B 0,C 180,E1 -23556.18,E2 -23556.18} C_VEL
LIN {X 0,Y 202.051,Z 336.081,A -85,B 0,C 180,E1 -23559.643,E2 -23559.643} C_VEL
LIN {X 0,Y 199.51,Z 333.003,A -85,B 0,C 180,E1 -23563.629,E2 -23563.629} C_VEL
LIN {X 0,Y 198.817,Z 331.129,A -85,B 0,C 180,E1 -23565.334,E2 -23565.334} C_VEL
LIN {X 0,Y 197.094,Z 329.817,A -85,B 0,C 180,E1 -23571.797,E2 -23571.797} C_VEL
LIN {X 0,Y 198.199,Z 330.418,A -85,B 0,C 180,E1 -23579.489,E2 -23579.489} C_VEL
LIN {X 0,Y 199.063,Z 331.239,A -85,B 0,C 180,E1 -23581.603,E2 -23581.603} C_VEL
LIN {X 0,Y 200.661,Z 334.332,A -85,B 0,C 180,E1 -23584.784,E2 -23584.784} C_VEL
LIN {X 0,Y 202.368,Z 336.333,A -85,B 0,C 180,E1 -23587.177,E2 -23587.177} C_VEL
LIN {X 0,Y 205.054,Z 340.318,A -85,B 0,C 180,E1 -23590.301,E2 -23590.301} C_VEL
LIN {X 0,Y 208.646,Z 345.727,A -85,B 0,C 180,E1 -23593.699,E2 -23593.699} C_VEL
LIN {X 0,Y 211.963,Z 350.853,A -85,B 0,C 180,E1 -23596.352,E2 -23596.352} C_VEL
LIN {X 0,Y 216.221,Z 357.805,A -85,B 0,C 180,E1 -23599.297,E2 -23599.297} C_VEL
LIN {X 0,Y 220.39,Z 365.22,A -85,B 0,C 180,E1 -23601.841,E2 -23601.841} C_VEL
LIN {X 0,Y 223.43,Z 371.851,A -85,B 0,C 180,E1 -23603.598,E2 -23603.598} C_VEL
LIN {X 0,Y 219.763,Z 415.135,A -85,B 0,C 180,E1 -23604.8,E2 -23604.8} C_VEL
LIN {X 0,Y 217.441,Z 429.708,A -85,B 0,C 180,E1 -23605.451,E2 -23605.451} C_VEL
LIN {X 0,Y 214.215,Z 443.543,A -85,B 0,C 180,E1 -23606.356,E2 -23606.356} C_VEL
LIN {X 0,Y 210.118,Z 457.021,A -85,B 0,C 180,E1 -23607.585,E2 -23607.585} C_VEL
LIN {X 0,Y 205.249,Z 469.988,A -85,B 0,C 180,E1 -23609.175,E2 -23609.175} C_VEL
LIN {X 0,Y 199.943,Z 481.732,A -85,B 0,C 180,E1 -23611.045,E2 -23611.045} C_VEL
LIN {X 0,Y 194.467,Z 492.018,A -85,B 0,C 180,E1 -23613.117,E2 -23613.117} C_VEL
LIN {X 0,Y 188.308,Z 502.161,A -85,B 0,C 180,E1 -23615.735,E2 -23615.735} C_VEL
LIN {X 0,Y 182.129,Z 511.126,A -85,B 0,C 180,E1 -23618.749,E2 -23618.749} C_VEL
LIN {X 0,Y 175.881,Z 519.221,A -85,B 0,C 180,E1 -23622.337,E2 -23622.337} C_VEL
LIN {X 0,Y 171.05,Z 524.99,A -85,B 0,C 180,E1 -23625.696,E2 -23625.696} C_VEL
LIN {X 0,Y 166.636,Z 529.847,A -85,B 0,C 180,E1 -23629.385,E2 -23629.385} C_VEL
LIN {X 0,Y 163.192,Z 533.306,A -85,B 0,C 180,E1 -23632.922,E2 -23632.922} C_VEL
LIN {X 0,Y 159.388,Z 536.792,A -85,B 0,C 180,E1 -23638.055,E2 -23638.055} C_VEL
LIN {X 0,Y 156.702,Z 538.759,A -85,B 0,C 180,E1 -23643.354,E2 -23643.354} C_VEL
LIN {X 0,Y 155.073,Z 539.265,A -85,B 0,C 180,E1 -23648.743,E2 -23648.743} C_VEL
LIN {X 0,Y 154.437,Z 538.368,A -85,B 0,C 180,E1 -23654.155,E2 -23654.155} C_VEL
LIN {X 0,Y 154.413,Z 536.091,A -85,B 0,C 180,E1 -23659.511,E2 -23659.511} C_VEL
LIN {X 0,Y 155.242,Z 532.387,A -85,B 0,C 180,E1 -23664.806,E2 -23664.806} C_VEL
LIN {X 0,Y 156.137,Z 528.63,A -85,B 0,C 180,E1 -23668.711,E2 -23668.711} C_VEL
LIN {X 0,Y 157.538,Z 523.972,A -85,B 0,C 180,E1 -23672.557,E2 -23672.557} C_VEL
LIN {X 0,Y 159.871,Z 517.193,A -85,B 0,C 180,E1 -23676.944,E2 -23676.944} C_VEL
LIN {X 0,Y 162.477,Z 510.112,A -85,B 0,C 180,E1 -23680.593,E2 -23680.593} C_VEL
LIN {X 0,Y 165.689,Z 501.592,A -85,B 0,C 180,E1 -23684.117,E2 -23684.117} C_VEL
LIN {X 0,Y 169.289,Z 491.654,A -85,B 0,C 180,E1 -23687.398,E2 -23687.398} C_VEL
LIN {X 0,Y 172.914,Z 480.921,A -85,B 0,C 180,E1 -23690.211,E2 -23690.211} C_VEL
LIN {X 0,Y 176.241,Z 469.696,A -85,B 0,C 180,E1 -23692.57,E2 -23692.57} C_VEL
LIN {X 0,Y 178.891,Z 459.217,A -85,B 0,C 180,E1 -23694.362,E2 -23694.362} C_VEL
LIN {X 0,Y 182.009,Z 446.066,A -85,B 0,C 180,E1 -23696.054,E2 -23696.054} C_VEL
LIN {X 0,Y 184.407,Z 431.831,A -85,B 0,C 180,E1 -23697.445,E2 -23697.445} C_VEL
LIN {X 0,Y 186.174,Z 417.646,A -85,B 0,C 180,E1 -23698.386,E2 -23698.386} C_VEL
LIN {X 0,Y 187.551,Z 398.199,A -85,B 0,C 180,E1 -23699.152,E2 -23699.152} C_VEL
LIN {X 0,Y 190.813,Z 345.483,A -85,B 0,C 180,E1 -23700.907,E2 -23700.907} C_VEL
LIN {X 0,Y 188.158,Z 338.72,A -85,B 0,C 180,E1 -23701.906,E2 -23701.906} C_VEL
LIN {X 0,Y 181.217,Z 325.078,A -85,B 0,C 180,E1 -23704.516,E2 -23704.516} C_VEL
LIN {X 0,Y 174.665,Z 313.956,A -85,B 0,C 180,E1 -23707.171,E2 -23707.171} C_VEL
LIN {X 0,Y 168.825,Z 305.236,A -85,B 0,C 180,E1 -23709.757,E2 -23709.757} C_VEL
LIN {X 0,Y 166.504,Z 301.953,A -85,B 0,C 180,E1 -23710.861,E2 -23710.861} C_VEL
LIN {X 0,Y 163.873,Z 298.191,A -85,B 0,C 180,E1 -23712.186,E2 -23712.186} C_VEL
LIN {X 0,Y 161.601,Z 295.183,A -85,B 0,C 180,E1 -23713.379,E2 -23713.379} C_VEL
LIN {X 0,Y 160.779,Z 293.77,A -85,B 0,C 180,E1 -23713.848,E2 -23713.848} C_VEL
LIN {X 0,Y 158.461,Z 291.637,A -85,B 0,C 180,E1 -23715.084,E2 -23715.084} C_VEL
LIN {X 0,Y 157.411,Z 289.116,A -85,B 0,C 180,E1 -23715.787,E2 -23715.787} C_VEL
LIN {X 0,Y 157.3,Z 288.492,A -85,B 0,C 180,E1 -23715.979,E2 -23715.979} C_VEL
LIN {X 0,Y 157.284,Z 288.511,A -85,B 0,C 180,E1 -23721.281,E2 -23721.281} C_VEL
LIN {X 0,Y 157.287,Z 288.484,A -85,B 0,C 180,E1 -23724.493,E2 -23724.493} C_VEL
LIN {X 0,Y 157.295,Z 288.514,A -85,B 0,C 180,E1 -23728.094,E2 -23728.094} C_VEL
LIN {X 0,Y 157.31,Z 288.477,A -85,B 0,C 180,E1 -23733.468,E2 -23733.468} C_VEL
LIN {X 0,Y 157.388,Z 288.498,A -85,B 0,C 180,E1 -23739.671,E2 -23739.671} C_VEL
LIN {X 0,Y 157.437,Z 288.492,A -85,B 0,C 180,E1 -23744.468,E2 -23744.468} C_VEL
LIN {X 0,Y 157.685,Z 288.457,A -85,B 0,C 180,E1 -23749.734,E2 -23749.734} C_VEL
LIN {X 0,Y 157.764,Z 288.42,A -85,B 0,C 180,E1 -23752.323,E2 -23752.323} C_VEL
LIN {X 0,Y 158.254,Z 288.385,A -85,B 0,C 180,E1 -23760.003,E2 -23760.003} C_VEL
LIN {X 0,Y 157.766,Z 288.458,A -85,B 0,C 180,E1 -23767.683,E2 -23767.683} C_VEL
LIN {X 0,Y 157.633,Z 288.445,A -85,B 0,C 180,E1 -23771.234,E2 -23771.234} C_VEL
LIN {X 0,Y 157.441,Z 288.49,A -85,B 0,C 180,E1 -23775.539,E2 -23775.539} C_VEL
LIN {X 0,Y 157.368,Z 288.508,A -85,B 0,C 180,E1 -23780.936,E2 -23780.936} C_VEL
LIN {X 0,Y 157.312,Z 288.51,A -85,B 0,C 180,E1 -23786.684,E2 -23786.684} C_VEL
LIN {X 0,Y 157.285,Z 288.518,A -85,B 0,C 180,E1 -23789.72,E2 -23789.72} C_VEL
LIN {X 0,Y 158.277,Z 291.294,A -85,B 0,C 180,E1 -23790.433,E2 -23790.433} C_VEL
LIN {X 0,Y 160.585,Z 293.614,A -85,B 0,C 180,E1 -23791.684,E2 -23791.684} C_VEL
LIN {X 0,Y 163.216,Z 297.585,A -85,B 0,C 180,E1 -23793.118,E2 -23793.118} C_VEL
LIN {X 0,Y 164.732,Z 299.383,A -85,B 0,C 180,E1 -23793.873,E2 -23793.873} C_VEL
LIN {X 0,Y 171.119,Z 308.651,A -85,B 0,C 180,E1 -23796.915,E2 -23796.915} C_VEL
LIN {X 0,Y 174.601,Z 314.229,A -85,B 0,C 180,E1 -23798.447,E2 -23798.447} C_VEL
LIN {X 0,Y 181.111,Z 327.7,A -85,B 0,C 180,E1 -23801.221,E2 -23801.221} C_VEL
LIN {X 0,Y 186.162,Z 339.914,A -85,B 0,C 180,E1 -23803.256,E2 -23803.256} C_VEL
LIN {X 0,Y 190.542,Z 352.608,A -85,B 0,C 180,E1 -23804.995,E2 -23804.995} C_VEL
LIN {X 0,Y 186.332,Z 422.64,A -85,B 0,C 180,E1 -23807.425,E2 -23807.425} C_VEL
LIN {X 0,Y 184.529,Z 437.372,A -85,B 0,C 180,E1 -23808.294,E2 -23808.294} C_VEL
LIN {X 0,Y 181.975,Z 451.407,A -85,B 0,C 180,E1 -23809.511,E2 -23809.511} C_VEL
LIN {X 0,Y 178.973,Z 464.472,A -85,B 0,C 180,E1 -23811.076,E2 -23811.076} C_VEL
LIN {X 0,Y 175.627,Z 477.217,A -85,B 0,C 180,E1 -23813.122,E2 -23813.122} C_VEL
LIN {X 0,Y 174.137,Z 480.554,A -85,B 0,C 180,E1 -23813.644,E2 -23813.644} C_VEL
LIN {X 0,Y 170.044,Z 485.633,A -85,B 0,C 180,E1 -23814.233,E2 -23814.233} C_VEL
LIN {X 0,Y 165.843,Z 490.606,A -85,B 0,C 180,E1 -23814.915,E2 -23814.915} C_VEL
LIN {X 0,Y 164.202,Z 493.637,A -85,B 0,C 180,E1 -23815.59,E2 -23815.59} C_VEL
LIN {X 0,Y 160.705,Z 503.048,A -85,B 0,C 180,E1 -23818.347,E2 -23818.347} C_VEL
LIN {X 0,Y 156.958,Z 512.865,A -85,B 0,C 180,E1 -23821.956,E2 -23821.956} C_VEL
LIN {X 0,Y 153.881,Z 520.99,A -85,B 0,C 180,E1 -23825.73,E2 -23825.73} C_VEL
LIN {X 0,Y 151.116,Z 528.763,A -85,B 0,C 180,E1 -23830.295,E2 -23830.295} C_VEL
LIN {X 0,Y 149.134,Z 534.959,A -85,B 0,C 180,E1 -23834.978,E2 -23834.978} C_VEL
LIN {X 0,Y 148.199,Z 539.161,A -85,B 0,C 180,E1 -23839.065,E2 -23839.065} C_VEL
LIN {X 0,Y 147.84,Z 541.462,A -85,B 0,C 180,E1 -23841.801,E2 -23841.801} C_VEL
LIN {X 0,Y 147.616,Z 544.919,A -85,B 0,C 180,E1 -23847.271,E2 -23847.271} C_VEL
LIN {X 0,Y 147.728,Z 546.104,A -85,B 0,C 180,E1 -23850,E2 -23850} C_VEL
LIN {X 0,Y 147.615,Z 546.928,A -85,B 0,C 180,E1 -23852.729,E2 -23852.729} C_VEL
LIN {X 0,Y 147.815,Z 547.57,A -85,B 0,C 180,E1 -23858.2,E2 -23858.2} C_VEL
LIN {X 0,Y 148.971,Z 546.907,A -85,B 0,C 180,E1 -23863.643,E2 -23863.643} C_VEL
LIN {X 0,Y 151.299,Z 544.943,A -85,B 0,C 180,E1 -23868.974,E2 -23868.974} C_VEL
LIN {X 0,Y 154.843,Z 541.628,A -85,B 0,C 180,E1 -23874.109,E2 -23874.109} C_VEL
LIN {X 0,Y 159.489,Z 536.869,A -85,B 0,C 180,E1 -23878.993,E2 -23878.993} C_VEL
LIN {X 0,Y 165.351,Z 530.529,A -85,B 0,C 180,E1 -23883.541,E2 -23883.541} C_VEL
LIN {X 0,Y 171.304,Z 523.511,A -85,B 0,C 180,E1 -23887.238,E2 -23887.238} C_VEL
LIN {X 0,Y 178.05,Z 514.854,A -85,B 0,C 180,E1 -23890.637,E2 -23890.637} C_VEL
LIN {X 0,Y 184.717,Z 505.114,A -85,B 0,C 180,E1 -23893.56,E2 -23893.56} C_VEL
LIN {X 0,Y 190.806,Z 494.966,A -85,B 0,C 180,E1 -23895.908,E2 -23895.908} C_VEL
LIN {X 0,Y 196.703,Z 483.926,A -85,B 0,C 180,E1 -23897.847,E2 -23897.847} C_VEL
LIN {X 0,Y 202.119,Z 471.811,A -85,B 0,C 180,E1 -23899.518,E2 -23899.518} C_VEL
LIN {X 0,Y 207.206,Z 458.229,A -85,B 0,C 180,E1 -23900.882,E2 -23900.882} C_VEL
LIN {X 0,Y 211.035,Z 445.098,A -85,B 0,C 180,E1 -23901.883,E2 -23901.883} C_VEL
LIN {X 0,Y 214.158,Z 430.835,A -85,B 0,C 180,E1 -23902.638,E2 -23902.638} C_VEL
LIN {X 0,Y 216.118,Z 416.618,A -85,B 0,C 180,E1 -23903.151,E2 -23903.151} C_VEL
LIN {X 0,Y 219.095,Z 380.75,A -85,B 0,C 180,E1 -23904.161,E2 -23904.161} C_VEL
LIN {X 0,Y 215.218,Z 371.147,A -85,B 0,C 180,E1 -23906.685,E2 -23906.685} C_VEL
LIN {X 0,Y 210.513,Z 360.865,A -85,B 0,C 180,E1 -23910.128,E2 -23910.128} C_VEL
LIN {X 0,Y 206.215,Z 352.43,A -85,B 0,C 180,E1 -23913.867,E2 -23913.867} C_VEL
LIN {X 0,Y 203.207,Z 347.149,A -85,B 0,C 180,E1 -23916.993,E2 -23916.993} C_VEL
LIN {X 0,Y 200.648,Z 342.769,A -85,B 0,C 180,E1 -23920.273,E2 -23920.273} C_VEL
LIN {X 0,Y 198.337,Z 339.733,A -85,B 0,C 180,E1 -23924.185,E2 -23924.185} C_VEL
LIN {X 0,Y 197.803,Z 338.181,A -85,B 0,C 180,E1 -23925.596,E2 -23925.596} C_VEL
LIN {X 0,Y 196.218,Z 336.873,A -85,B 0,C 180,E1 -23931.76,E2 -23931.76} C_VEL
LIN {X 0,Y 197.138,Z 337.34,A -85,B 0,C 180,E1 -23938.976,E2 -23938.976} C_VEL
LIN {X 0,Y 197.985,Z 338.131,A -85,B 0,C 180,E1 -23941.192,E2 -23941.192} C_VEL
LIN {X 0,Y 199.526,Z 341.226,A -85,B 0,C 180,E1 -23944.424,E2 -23944.424} C_VEL
LIN {X 0,Y 201.027,Z 343.074,A -85,B 0,C 180,E1 -23946.647,E2 -23946.647} C_VEL
LIN {X 0,Y 203.741,Z 347.168,A -85,B 0,C 180,E1 -23949.929,E2 -23949.929} C_VEL
LIN {X 0,Y 206.929,Z 352.246,A -85,B 0,C 180,E1 -23953.081,E2 -23953.081} C_VEL
LIN {X 0,Y 211.023,Z 358.819,A -85,B 0,C 180,E1 -23956.442,E2 -23956.442} C_VEL
LIN {X 0,Y 215.232,Z 366.185,A -85,B 0,C 180,E1 -23959.392,E2 -23959.392} C_VEL
LIN {X 0,Y 218.536,Z 372.637,A -85,B 0,C 180,E1 -23961.474,E2 -23961.474} C_VEL
LIN {X 0,Y 219.563,Z 375.04,A -85,B 0,C 180,E1 -23962.107,E2 -23962.107} C_VEL
LIN {X 0,Y 215.955,Z 415.792,A -85,B 0,C 180,E1 -23963.237,E2 -23963.237} C_VEL
LIN {X 0,Y 213.535,Z 430.35,A -85,B 0,C 180,E1 -23963.889,E2 -23963.889} C_VEL
LIN {X 0,Y 210.375,Z 443.48,A -85,B 0,C 180,E1 -23964.739,E2 -23964.739} C_VEL
LIN {X 0,Y 206.155,Z 457.01,A -85,B 0,C 180,E1 -23965.957,E2 -23965.957} C_VEL
LIN {X 0,Y 201.049,Z 470.142,A -85,B 0,C 180,E1 -23967.547,E2 -23967.547} C_VEL
LIN {X 0,Y 195.612,Z 481.793,A -85,B 0,C 180,E1 -23969.397,E2 -23969.397} C_VEL
LIN {X 0,Y 189.685,Z 492.515,A -85,B 0,C 180,E1 -23971.554,E2 -23971.554} C_VEL
LIN {X 0,Y 184.01,Z 501.426,A -85,B 0,C 180,E1 -23973.831,E2 -23973.831} C_VEL
LIN {X 0,Y 177.986,Z 510.004,A -85,B 0,C 180,E1 -23976.654,E2 -23976.654} C_VEL
LIN {X 0,Y 171.868,Z 517.748,A -85,B 0,C 180,E1 -23979.942,E2 -23979.942} C_VEL
LIN {X 0,Y 165.749,Z 524.72,A -85,B 0,C 180,E1 -23983.879,E2 -23983.879} C_VEL
LIN {X 0,Y 160.513,Z 530.154,A -85,B 0,C 180,E1 -23988.097,E2 -23988.097} C_VEL
LIN {X 0,Y 157.251,Z 533.196,A -85,B 0,C 180,E1 -23991.268,E2 -23991.268} C_VEL
LIN {X 0,Y 153.058,Z 536.781,A -85,B 0,C 180,E1 -23996.565,E2 -23996.565} C_VEL
LIN {X 0,Y 150.06,Z 538.862,A -85,B 0,C 180,E1 -24002.074,E2 -24002.074} C_VEL
LIN {X 0,Y 148.181,Z 539.495,A -85,B 0,C 180,E1 -24007.703,E2 -24007.703} C_VEL
LIN {X 0,Y 147.405,Z 538.692,A -85,B 0,C 180,E1 -24013.378,E2 -24013.378} C_VEL
LIN {X 0,Y 147.281,Z 536.508,A -85,B 0,C 180,E1 -24018.997,E2 -24018.997} C_VEL
LIN {X 0,Y 148.059,Z 532.9,A -85,B 0,C 180,E1 -24024.553,E2 -24024.553} C_VEL
LIN {X 0,Y 149,Z 529.242,A -85,B 0,C 180,E1 -24028.649,E2 -24028.649} C_VEL
LIN {X 0,Y 150.436,Z 524.646,A -85,B 0,C 180,E1 -24032.678,E2 -24032.678} C_VEL
LIN {X 0,Y 152.814,Z 518.007,A -85,B 0,C 180,E1 -24037.266,E2 -24037.266} C_VEL
LIN {X 0,Y 156.018,Z 509.745,A -85,B 0,C 180,E1 -24041.695,E2 -24041.695} C_VEL
LIN {X 0,Y 159.414,Z 501.112,A -85,B 0,C 180,E1 -24045.338,E2 -24045.338} C_VEL
LIN {X 0,Y 163.23,Z 491.036,A -85,B 0,C 180,E1 -24048.709,E2 -24048.709} C_VEL
LIN {X 0,Y 167.019,Z 480.124,A -85,B 0,C 180,E1 -24051.604,E2 -24051.604} C_VEL
LIN {X 0,Y 170.844,Z 467.286,A -85,B 0,C 180,E1 -24054.291,E2 -24054.291} C_VEL
LIN {X 0,Y 173.805,Z 456.176,A -85,B 0,C 180,E1 -24056.087,E2 -24056.087} C_VEL
LIN {X 0,Y 176.553,Z 444.359,A -85,B 0,C 180,E1 -24057.564,E2 -24057.564} C_VEL
LIN {X 0,Y 178.961,Z 430.217,A -85,B 0,C 180,E1 -24058.916,E2 -24058.916} C_VEL
LIN {X 0,Y 180.702,Z 416.26,A -85,B 0,C 180,E1 -24059.808,E2 -24059.808} C_VEL
LIN {X 0,Y 182.548,Z 389.882,A -85,B 0,C 180,E1 -24060.788,E2 -24060.788} C_VEL
LIN {X 0,Y 185.284,Z 347.472,A -85,B 0,C 180,E1 -24062.218,E2 -24062.218} C_VEL
LIN {X 0,Y 182.863,Z 341.549,A -85,B 0,C 180,E1 -24063.178,E2 -24063.178} C_VEL
LIN {X 0,Y 176.55,Z 329.02,A -85,B 0,C 180,E1 -24065.705,E2 -24065.705} C_VEL
LIN {X 0,Y 170.198,Z 318.184,A -85,B 0,C 180,E1 -24068.452,E2 -24068.452} C_VEL
LIN {X 0,Y 163.675,Z 308.138,A -85,B 0,C 180,E1 -24071.593,E2 -24071.593} C_VEL
LIN {X 0,Y 160.088,Z 303.285,A -85,B 0,C 180,E1 -24073.478,E2 -24073.478} C_VEL
LIN {X 0,Y 157.424,Z 299.519,A -85,B 0,C 180,E1 -24074.992,E2 -24074.992} C_VEL
LIN {X 0,Y 155.077,Z 296.796,A -85,B 0,C 180,E1 -24076.368,E2 -24076.368} C_VEL
LIN {X 0,Y 153.882,Z 294.7,A -85,B 0,C 180,E1 -24077.161,E2 -24077.161} C_VEL
LIN {X 0,Y 151.619,Z 292.796,A -85,B 0,C 180,E1 -24078.565,E2 -24078.565} C_VEL
LIN {X 0,Y 150.41,Z 290.301,A -85,B 0,C 180,E1 -24079.481,E2 -24079.481} C_VEL
LIN {X 0,Y 150.25,Z 289.39,A -85,B 0,C 180,E1 -24079.758,E2 -24079.758} C_VEL
LIN {X 0,Y 150.231,Z 289.369,A -85,B 0,C 180,E1 -24082.681,E2 -24082.681} C_VEL
LIN {X 0,Y 150.217,Z 289.39,A -85,B 0,C 180,E1 -24087.366,E2 -24087.366} C_VEL
LIN {X 0,Y 150.236,Z 289.357,A -85,B 0,C 180,E1 -24092.723,E2 -24092.723} C_VEL
LIN {X 0,Y 150.346,Z 289.377,A -85,B 0,C 180,E1 -24099.212,E2 -24099.212} C_VEL
LIN {X 0,Y 150.349,Z 289.38,A -85,B 0,C 180,E1 -24103.716,E2 -24103.716} C_VEL
LIN {X 0,Y 150.607,Z 289.344,A -85,B 0,C 180,E1 -24109.246,E2 -24109.246} C_VEL
LIN {X 0,Y 150.685,Z 289.302,A -85,B 0,C 180,E1 -24111.96,E2 -24111.96} C_VEL
LIN {X 0,Y 151.215,Z 289.261,A -85,B 0,C 180,E1 -24120.004,E2 -24120.004} C_VEL
LIN {X 0,Y 150.703,Z 289.339,A -85,B 0,C 180,E1 -24128.046,E2 -24128.046} C_VEL
LIN {X 0,Y 150.575,Z 289.321,A -85,B 0,C 180,E1 -24131.436,E2 -24131.436} C_VEL
LIN {X 0,Y 150.353,Z 289.379,A -85,B 0,C 180,E1 -24136.291,E2 -24136.291} C_VEL
LIN {X 0,Y 150.351,Z 289.38,A -85,B 0,C 180,E1 -24140.794,E2 -24140.794} C_VEL
LIN {X 0,Y 150.239,Z 289.395,A -85,B 0,C 180,E1 -24145.954,E2 -24145.954} C_VEL
LIN {X 0,Y 151.126,Z 292.003,A -85,B 0,C 180,E1 -24146.712,E2 -24146.712} C_VEL
LIN {X 0,Y 152.942,Z 294.158,A -85,B 0,C 180,E1 -24147.917,E2 -24147.917} C_VEL
LIN {X 0,Y 154.332,Z 295.277,A -85,B 0,C 180,E1 -24148.754,E2 -24148.754} C_VEL
LIN {X 0,Y 156.296,Z 298.382,A -85,B 0,C 180,E1 -24150.001,E2 -24150.001} C_VEL
LIN {X 0,Y 158.006,Z 300.328,A -85,B 0,C 180,E1 -24150.978,E2 -24150.978} C_VEL
LIN {X 0,Y 160.577,Z 303.898,A -85,B 0,C 180,E1 -24152.414,E2 -24152.414} C_VEL
LIN {X 0,Y 164.868,Z 310.141,A -85,B 0,C 180,E1 -24154.646,E2 -24154.646} C_VEL
LIN {X 0,Y 170.248,Z 318.394,A -85,B 0,C 180,E1 -24157.199,E2 -24157.199} C_VEL
LIN {X 0,Y 176.64,Z 332.032,A -85,B 0,C 180,E1 -24160.116,E2 -24160.116} C_VEL
LIN {X 0,Y 181.573,Z 344.367,A -85,B 0,C 180,E1 -24162.236,E2 -24162.236} C_VEL
LIN {X 0,Y 184.996,Z 354.434,A -85,B 0,C 180,E1 -24163.682,E2 -24163.682} C_VEL
LIN {X 0,Y 180.733,Z 422.117,A -85,B 0,C 180,E1 -24166.063,E2 -24166.063} C_VEL
LIN {X 0,Y 178.86,Z 436.972,A -85,B 0,C 180,E1 -24166.944,E2 -24166.944} C_VEL
LIN {X 0,Y 176.327,Z 450.486,A -85,B 0,C 180,E1 -24168.117,E2 -24168.117} C_VEL
LIN {X 0,Y 173.514,Z 462.837,A -85,B 0,C 180,E1 -24169.605,E2 -24169.605} C_VEL
LIN {X 0,Y 170.354,Z 474.352,A -85,B 0,C 180,E1 -24171.393,E2 -24171.393} C_VEL
LIN {X 0,Y 166.745,Z 486.414,A -85,B 0,C 180,E1 -24173.838,E2 -24173.838} C_VEL
LIN {X 0,Y 164.202,Z 493.637,A -85,B 0,C 180,E1 -24175.59,E2 -24175.59} C_VEL
LIN {X 0,Y 162.078,Z 498.112,A -85,B 0,C 180,E1 -24176.719,E2 -24176.719} C_VEL
LIN {X 0,Y 156.874,Z 505.023,A -85,B 0,C 180,E1 -24178.463,E2 -24178.463} C_VEL
LIN {X 0,Y 151.602,Z 511.44,A -85,B 0,C 180,E1 -24180.487,E2 -24180.487} C_VEL
LIN {X 0,Y 149.436,Z 515.143,A -85,B 0,C 180,E1 -24182.036,E2 -24182.036} C_VEL
LIN {X 0,Y 146.015,Z 523.49,A -85,B 0,C 180,E1 -24186.366,E2 -24186.366} C_VEL
LIN {X 0,Y 144.023,Z 529.163,A -85,B 0,C 180,E1 -24190.027,E2 -24190.027} C_VEL
LIN {X 0,Y 142.245,Z 534.428,A -85,B 0,C 180,E1 -24194.232,E2 -24194.232} C_VEL
LIN {X 0,Y 141.183,Z 538.705,A -85,B 0,C 180,E1 -24198.515,E2 -24198.515} C_VEL
LIN {X 0,Y 140.793,Z 541.045,A -85,B 0,C 180,E1 -24201.387,E2 -24201.387} C_VEL
LIN {X 0,Y 140.513,Z 544.571,A -85,B 0,C 180,E1 -24207.133,E2 -24207.133} C_VEL
LIN {X 0,Y 140.594,Z 546.175,A -85,B 0,C 180,E1 -24211.108,E2 -24211.108} C_VEL
LIN {X 0,Y 140.542,Z 547.165,A -85,B 0,C 180,E1 -24215.739,E2 -24215.739} C_VEL
LIN {X 0,Y 141.297,Z 547.217,A -85,B 0,C 180,E1 -24221.475,E2 -24221.475} C_VEL
LIN {X 0,Y 143.087,Z 545.974,A -85,B 0,C 180,E1 -24227.139,E2 -24227.139} C_VEL
LIN {X 0,Y 146.3,Z 543.428,A -85,B 0,C 180,E1 -24232.6,E2 -24232.6} C_VEL
LIN {X 0,Y 150.626,Z 539.499,A -85,B 0,C 180,E1 -24237.812,E2 -24237.812} C_VEL
LIN {X 0,Y 156.256,Z 534.051,A -85,B 0,C 180,E1 -24242.664,E2 -24242.664} C_VEL
LIN {X 0,Y 161.193,Z 528.909,A -85,B 0,C 180,E1 -24246.056,E2 -24246.056} C_VEL
LIN {X 0,Y 167.671,Z 521.556,A -85,B 0,C 180,E1 -24249.731,E2 -24249.731} C_VEL
LIN {X 0,Y 174.867,Z 512.454,A -85,B 0,C 180,E1 -24253.096,E2 -24253.096} C_VEL
LIN {X 0,Y 181.459,Z 502.785,A -85,B 0,C 180,E1 -24255.861,E2 -24255.861} C_VEL
LIN {X 0,Y 187.76,Z 492.533,A -85,B 0,C 180,E1 -24258.066,E2 -24258.066} C_VEL
LIN {X 0,Y 193.875,Z 481.008,A -85,B 0,C 180,E1 -24259.975,E2 -24259.975} C_VEL
LIN {X 0,Y 198.906,Z 469.816,A -85,B 0,C 180,E1 -24261.419,E2 -24261.419} C_VEL
LIN {X 0,Y 203.502,Z 457.74,A -85,B 0,C 180,E1 -24262.588,E2 -24262.588} C_VEL
LIN {X 0,Y 207.451,Z 444.517,A -85,B 0,C 180,E1 -24263.569,E2 -24263.569} C_VEL
LIN {X 0,Y 210.58,Z 430.557,A -85,B 0,C 180,E1 -24264.288,E2 -24264.288} C_VEL
LIN {X 0,Y 212.568,Z 416.461,A -85,B 0,C 180,E1 -24264.794,E2 -24264.794} C_VEL
LIN {X 0,Y 215.41,Z 383.848,A -85,B 0,C 180,E1 -24265.69,E2 -24265.69} C_VEL
LIN {X 0,Y 212.14,Z 375.611,A -85,B 0,C 180,E1 -24267.988,E2 -24267.988} C_VEL
LIN {X 0,Y 208.272,Z 366.707,A -85,B 0,C 180,E1 -24271.054,E2 -24271.054} C_VEL
LIN {X 0,Y 204.356,Z 358.648,A -85,B 0,C 180,E1 -24274.685,E2 -24274.685} C_VEL
LIN {X 0,Y 201.503,Z 353.381,A -85,B 0,C 180,E1 -24277.858,E2 -24277.858} C_VEL
LIN {X 0,Y 199.562,Z 349.76,A -85,B 0,C 180,E1 -24280.502,E2 -24280.502} C_VEL
LIN {X 0,Y 197.217,Z 346.532,A -85,B 0,C 180,E1 -24284.666,E2 -24284.666} C_VEL
LIN {X 0,Y 196.669,Z 345.069,A -85,B 0,C 180,E1 -24286.187,E2 -24286.187} C_VEL
LIN {X 0,Y 195.341,Z 343.93,A -85,B 0,C 180,E1 -24291.723,E2 -24291.723} C_VEL
LIN {X 0,Y 196.252,Z 344.395,A -85,B 0,C 180,E1 -24298.971,E2 -24298.971} C_VEL
LIN {X 0,Y 196.918,Z 345.081,A -85,B 0,C 180,E1 -24300.794,E2 -24300.794} C_VEL
LIN {X 0,Y 198.513,Z 348.253,A -85,B 0,C 180,E1 -24304.252,E2 -24304.252} C_VEL
LIN {X 0,Y 199.736,Z 349.9,A -85,B 0,C 180,E1 -24306.162,E2 -24306.162} C_VEL
LIN {X 0,Y 202.798,Z 354.788,A -85,B 0,C 180,E1 -24309.975,E2 -24309.975} C_VEL
LIN {X 0,Y 205.33,Z 358.98,A -85,B 0,C 180,E1 -24312.547,E2 -24312.547} C_VEL
LIN {X 0,Y 208.815,Z 364.703,A -85,B 0,C 180,E1 -24315.55,E2 -24315.55} C_VEL
LIN {X 0,Y 213.164,Z 372.703,A -85,B 0,C 180,E1 -24318.779,E2 -24318.779} C_VEL
LIN {X 0,Y 215.837,Z 378.28,A -85,B 0,C 180,E1 -24320.561,E2 -24320.561} C_VEL
LIN {X 0,Y 212.424,Z 415.701,A -85,B 0,C 180,E1 -24321.593,E2 -24321.593} C_VEL
LIN {X 0,Y 209.962,Z 430.198,A -85,B 0,C 180,E1 -24322.225,E2 -24322.225} C_VEL
LIN {X 0,Y 206.712,Z 443.42,A -85,B 0,C 180,E1 -24323.063,E2 -24323.063} C_VEL
LIN {X 0,Y 202.362,Z 457.006,A -85,B 0,C 180,E1 -24324.268,E2 -24324.268} C_VEL
LIN {X 0,Y 197.446,Z 469.352,A -85,B 0,C 180,E1 -24325.732,E2 -24325.732} C_VEL
LIN {X 0,Y 192.067,Z 480.631,A -85,B 0,C 180,E1 -24327.462,E2 -24327.462} C_VEL
LIN {X 0,Y 185.909,Z 491.587,A -85,B 0,C 180,E1 -24329.605,E2 -24329.605} C_VEL
LIN {X 0,Y 179.978,Z 500.685,A -85,B 0,C 180,E1 -24331.865,E2 -24331.865} C_VEL
LIN {X 0,Y 173.705,Z 509.31,A -85,B 0,C 180,E1 -24334.633,E2 -24334.633} C_VEL
LIN {X 0,Y 167.148,Z 517.302,A -85,B 0,C 180,E1 -24337.968,E2 -24337.968} C_VEL
LIN {X 0,Y 160.632,Z 524.408,A -85,B 0,C 180,E1 -24341.947,E2 -24341.947} C_VEL
LIN {X 0,Y 155.753,Z 529.248,A -85,B 0,C 180,E1 -24345.625,E2 -24345.625} C_VEL
LIN {X 0,Y 151.471,Z 533.093,A -85,B 0,C 180,E1 -24349.492,E2 -24349.492} C_VEL
LIN {X 0,Y 146.846,Z 536.778,A -85,B 0,C 180,E1 -24354.95,E2 -24354.95} C_VEL
LIN {X 0,Y 143.486,Z 538.953,A -85,B 0,C 180,E1 -24360.673,E2 -24360.673} C_VEL
LIN {X 0,Y 141.33,Z 539.692,A -85,B 0,C 180,E1 -24366.559,E2 -24366.559} C_VEL
LIN {X 0,Y 140.381,Z 539.013,A -85,B 0,C 180,E1 -24372.52,E2 -24372.52} C_VEL
LIN {X 0,Y 140.143,Z 536.926,A -85,B 0,C 180,E1 -24378.429,E2 -24378.429} C_VEL
LIN {X 0,Y 140.866,Z 533.414,A -85,B 0,C 180,E1 -24384.274,E2 -24384.274} C_VEL
LIN {X 0,Y 141.866,Z 529.845,A -85,B 0,C 180,E1 -24388.581,E2 -24388.581} C_VEL
LIN {X 0,Y 143.304,Z 525.313,A -85,B 0,C 180,E1 -24392.811,E2 -24392.811} C_VEL
LIN {X 0,Y 145.752,Z 518.788,A -85,B 0,C 180,E1 -24397.62,E2 -24397.62} C_VEL
LIN {X 0,Y 149.047,Z 510.696,A -85,B 0,C 180,E1 -24402.251,E2 -24402.251} C_VEL
LIN {X 0,Y 152.585,Z 502.21,A -85,B 0,C 180,E1 -24406.043,E2 -24406.043} C_VEL
LIN {X 0,Y 156.42,Z 492.62,A -85,B 0,C 180,E1 -24409.454,E2 -24409.454} C_VEL
LIN {X 0,Y 160.5,Z 481.57,A -85,B 0,C 180,E1 -24412.553,E2 -24412.553} C_VEL
LIN {X 0,Y 164.461,Z 469.088,A -85,B 0,C 180,E1 -24415.298,E2 -24415.298} C_VEL
LIN {X 0,Y 167.435,Z 458.382,A -85,B 0,C 180,E1 -24417.159,E2 -24417.159} C_VEL
LIN {X 0,Y 170.575,Z 445.963,A -85,B 0,C 180,E1 -24418.786,E2 -24418.786} C_VEL
LIN {X 0,Y 173.056,Z 432.311,A -85,B 0,C 180,E1 -24420.169,E2 -24420.169} C_VEL
LIN {X 0,Y 174.972,Z 418.155,A -85,B 0,C 180,E1 -24421.14,E2 -24421.14} C_VEL
LIN {X 0,Y 176.515,Z 397.995,A -85,B 0,C 180,E1 -24421.962,E2 -24421.962} C_VEL
LIN {X 0,Y 179.825,Z 349.382,A -85,B 0,C 180,E1 -24423.619,E2 -24423.619} C_VEL
LIN {X 0,Y 173.696,Z 336.27,A -85,B 0,C 180,E1 -24426.197,E2 -24426.197} C_VEL
LIN {X 0,Y 167.015,Z 324.262,A -85,B 0,C 180,E1 -24429.232,E2 -24429.232} C_VEL
LIN {X 0,Y 160.247,Z 313.578,A -85,B 0,C 180,E1 -24432.675,E2 -24432.675} C_VEL
LIN {X 0,Y 156.496,Z 308.422,A -85,B 0,C 180,E1 -24434.768,E2 -24434.768} C_VEL
LIN {X 0,Y 154.257,Z 305.214,A -85,B 0,C 180,E1 -24436.126,E2 -24436.126} C_VEL
LIN {X 0,Y 151.76,Z 301.959,A -85,B 0,C 180,E1 -24437.716,E2 -24437.716} C_VEL
LIN {X 0,Y 150.953,Z 300.767,A -85,B 0,C 180,E1 -24438.265,E2 -24438.265} C_VEL
LIN {X 0,Y 148.574,Z 298.253,A -85,B 0,C 180,E1 -24439.877,E2 -24439.877} C_VEL
LIN {X 0,Y 147.399,Z 295.882,A -85,B 0,C 180,E1 -24440.825,E2 -24440.825} C_VEL
LIN {X 0,Y 144.92,Z 294.082,A -85,B 0,C 180,E1 -24442.649,E2 -24442.649} C_VEL
LIN {X 0,Y 143.505,Z 291.836,A -85,B 0,C 180,E1 -24443.894,E2 -24443.894} C_VEL
LIN {X 0,Y 143.134,Z 290.244,A -85,B 0,C 180,E1 -24444.459,E2 -24444.459} C_VEL
LIN {X 0,Y 143.184,Z 290.263,A -85,B 0,C 180,E1 -24447.327,E2 -24447.327} C_VEL
LIN {X 0,Y 143.184,Z 290.237,A -85,B 0,C 180,E1 -24452.067,E2 -24452.067} C_VEL
LIN {X 0,Y 143.271,Z 290.261,A -85,B 0,C 180,E1 -24458.75,E2 -24458.75} C_VEL
LIN {X 0,Y 143.292,Z 290.262,A -85,B 0,C 180,E1 -24462.89,E2 -24462.89} C_VEL
LIN {X 0,Y 143.533,Z 290.228,A -85,B 0,C 180,E1 -24468.709,E2 -24468.709} C_VEL
LIN {X 0,Y 143.61,Z 290.185,A -85,B 0,C 180,E1 -24471.562,E2 -24471.562} C_VEL
LIN {X 0,Y 144.173,Z 290.135,A -85,B 0,C 180,E1 -24480.004,E2 -24480.004} C_VEL
LIN {X 0,Y 143.625,Z 290.218,A -85,B 0,C 180,E1 -24488.445,E2 -24488.445} C_VEL
LIN {X 0,Y 143.502,Z 290.2,A -85,B 0,C 180,E1 -24491.626,E2 -24491.626} C_VEL
LIN {X 0,Y 143.29,Z 290.262,A -85,B 0,C 180,E1 -24497.118,E2 -24497.118} C_VEL
LIN {X 0,Y 143.274,Z 290.438,A -85,B 0,C 180,E1 -24501.418,E2 -24501.418} C_VEL
LIN {X 0,Y 144.041,Z 292.844,A -85,B 0,C 180,E1 -24502.231,E2 -24502.231} C_VEL
LIN {X 0,Y 145.799,Z 294.966,A -85,B 0,C 180,E1 -24503.664,E2 -24503.664} C_VEL
LIN {X 0,Y 147.548,Z 296.162,A -85,B 0,C 180,E1 -24504.916,E2 -24504.916} C_VEL
LIN {X 0,Y 149.295,Z 299.222,A -85,B 0,C 180,E1 -24506.263,E2 -24506.263} C_VEL
LIN {X 0,Y 151.614,Z 301.62,A -85,B 0,C 180,E1 -24507.804,E2 -24507.804} C_VEL
LIN {X 0,Y 154.333,Z 305.27,A -85,B 0,C 180,E1 -24509.548,E2 -24509.548} C_VEL
LIN {X 0,Y 158.836,Z 311.768,A -85,B 0,C 180,E1 -24512.197,E2 -24512.197} C_VEL
LIN {X 0,Y 163.445,Z 318.571,A -85,B 0,C 180,E1 -24514.634,E2 -24514.634} C_VEL
LIN {X 0,Y 166.841,Z 324.437,A -85,B 0,C 180,E1 -24516.335,E2 -24516.335} C_VEL
LIN {X 0,Y 172.663,Z 337.363,A -85,B 0,C 180,E1 -24519.151,E2 -24519.151} C_VEL
LIN {X 0,Y 177.305,Z 349.553,A -85,B 0,C 180,E1 -24521.284,E2 -24521.284} C_VEL
LIN {X 0,Y 179.503,Z 356.279,A -85,B 0,C 180,E1 -24522.282,E2 -24522.282} C_VEL
LIN {X 0,Y 175.121,Z 422.754,A -85,B 0,C 180,E1 -24524.677,E2 -24524.677} C_VEL
LIN {X 0,Y 173.177,Z 437.315,A -85,B 0,C 180,E1 -24525.57,E2 -24525.57} C_VEL
LIN {X 0,Y 170.55,Z 450.69,A -85,B 0,C 180,E1 -24526.759,E2 -24526.759} C_VEL
LIN {X 0,Y 167.635,Z 462.959,A -85,B 0,C 180,E1 -24528.276,E2 -24528.276} C_VEL
LIN {X 0,Y 164.353,Z 474.417,A -85,B 0,C 180,E1 -24530.103,E2 -24530.103} C_VEL
LIN {X 0,Y 160.59,Z 486.438,A -85,B 0,C 180,E1 -24532.612,E2 -24532.612} C_VEL
LIN {X 0,Y 157.706,Z 494.326,A -85,B 0,C 180,E1 -24534.597,E2 -24534.597} C_VEL
LIN {X 0,Y 153.921,Z 503.921,A -85,B 0,C 180,E1 -24537.555,E2 -24537.555} C_VEL
LIN {X 0,Y 150.056,Z 513.562,A -85,B 0,C 180,E1 -24541.311,E2 -24541.311} C_VEL
LIN {X 0,Y 149.436,Z 515.143,A -85,B 0,C 180,E1 -24542.036,E2 -24542.036} C_VEL
LIN {X 0,Y 147.362,Z 518.739,A -85,B 0,C 180,E1 -24543.687,E2 -24543.687} C_VEL
LIN {X 0,Y 142.464,Z 524.092,A -85,B 0,C 180,E1 -24546.369,E2 -24546.369} C_VEL
LIN {X 0,Y 137.812,Z 528.956,A -85,B 0,C 180,E1 -24549.357,E2 -24549.357} C_VEL
LIN {X 0,Y 136.182,Z 531.635,A -85,B 0,C 180,E1 -24551.435,E2 -24551.435} C_VEL
LIN {X 0,Y 134.493,Z 536.907,A -85,B 0,C 180,E1 -24556.4,E2 -24556.4} C_VEL
LIN {X 0,Y 133.741,Z 540.623,A -85,B 0,C 180,E1 -24560.929,E2 -24560.929} C_VEL
LIN {X 0,Y 133.414,Z 544.221,A -85,B 0,C 180,E1 -24566.98,E2 -24566.98} C_VEL
LIN {X 0,Y 133.542,Z 545.598,A -85,B 0,C 180,E1 -24570.338,E2 -24570.338} C_VEL
LIN {X 0,Y 133.458,Z 546.913,A -85,B 0,C 180,E1 -24576.045,E2 -24576.045} C_VEL
LIN {X 0,Y 134.305,Z 547.033,A -85,B 0,C 180,E1 -24582.082,E2 -24582.082} C_VEL
LIN {X 0,Y 136.283,Z 545.859,A -85,B 0,C 180,E1 -24588.023,E2 -24588.023} C_VEL
LIN {X 0,Y 139.731,Z 543.382,A -85,B 0,C 180,E1 -24593.726,E2 -24593.726} C_VEL
LIN {X 0,Y 144.358,Z 539.54,A -85,B 0,C 180,E1 -24599.132,E2 -24599.132} C_VEL
LIN {X 0,Y 150.309,Z 534.195,A -85,B 0,C 180,E1 -24604.13,E2 -24604.13} C_VEL
LIN {X 0,Y 157.335,Z 527.164,A -85,B 0,C 180,E1 -24608.708,E2 -24608.708} C_VEL
LIN {X 0,Y 164.364,Z 519.44,A -85,B 0,C 180,E1 -24612.332,E2 -24612.332} C_VEL
LIN {X 0,Y 171.993,Z 509.935,A -85,B 0,C 180,E1 -24615.649,E2 -24615.649} C_VEL
LIN {X 0,Y 178.822,Z 500.02,A -85,B 0,C 180,E1 -24618.306,E2 -24618.306} C_VEL
LIN {X 0,Y 185.639,Z 488.989,A -85,B 0,C 180,E1 -24620.474,E2 -24620.474} C_VEL
LIN {X 0,Y 191.975,Z 476.694,A -85,B 0,C 180,E1 -24622.34,E2 -24622.34} C_VEL
LIN {X 0,Y 197.319,Z 464.523,A -85,B 0,C 180,E1 -24623.69,E2 -24623.69} C_VEL
LIN {X 0,Y 201.998,Z 451.062,A -85,B 0,C 180,E1 -24624.845,E2 -24624.845} C_VEL
LIN {X 0,Y 205.775,Z 437.07,A -85,B 0,C 180,E1 -24625.68,E2 -24625.68} C_VEL
LIN {X 0,Y 208.354,Z 423.266,A -85,B 0,C 180,E1 -24626.26,E2 -24626.26} C_VEL
LIN {X 0,Y 210.736,Z 399.641,A -85,B 0,C 180,E1 -24626.937,E2 -24626.937} C_VEL
LIN {X 0,Y 211.798,Z 386.899,A -85,B 0,C 180,E1 -24627.321,E2 -24627.321} C_VEL
LIN {X 0,Y 208.978,Z 379.464,A -85,B 0,C 180,E1 -24629.512,E2 -24629.512} C_VEL
LIN {X 0,Y 205.626,Z 371.618,A -85,B 0,C 180,E1 -24632.413,E2 -24632.413} C_VEL
LIN {X 0,Y 202.506,Z 364.758,A -85,B 0,C 180,E1 -24635.558,E2 -24635.558} C_VEL
LIN {X 0,Y 199.959,Z 359.845,A -85,B 0,C 180,E1 -24638.585,E2 -24638.585} C_VEL
LIN {X 0,Y 198.266,Z 356.544,A -85,B 0,C 180,E1 -24641.053,E2 -24641.053} C_VEL
LIN {X 0,Y 196.041,Z 353.172,A -85,B 0,C 180,E1 -24645.336,E2 -24645.336} C_VEL
LIN {X 0,Y 195.676,Z 352.071,A -85,B 0,C 180,E1 -24646.454,E2 -24646.454} C_VEL
LIN {X 0,Y 194.465,Z 350.986,A -85,B 0,C 180,E1 -24651.685,E2 -24651.685} C_VEL
LIN {X 0,Y 195.204,Z 351.352,A -85,B 0,C 180,E1 -24658.45,E2 -24658.45} C_VEL
LIN {X 0,Y 195.875,Z 352.046,A -85,B 0,C 180,E1 -24660.427,E2 -24660.427} C_VEL
LIN {X 0,Y 197.726,Z 355.607,A -85,B 0,C 180,E1 -24664.465,E2 -24664.465} C_VEL
LIN {X 0,Y 198.495,Z 356.737,A -85,B 0,C 180,E1 -24665.701,E2 -24665.701} C_VEL
LIN {X 0,Y 201.253,Z 361.379,A -85,B 0,C 180,E1 -24669.339,E2 -24669.339} C_VEL
LIN {X 0,Y 203.922,Z 365.929,A -85,B 0,C 180,E1 -24672.166,E2 -24672.166} C_VEL
LIN {X 0,Y 207.676,Z 372.597,A -85,B 0,C 180,E1 -24675.503,E2 -24675.503} C_VEL
LIN {X 0,Y 211.509,Z 380.025,A -85,B 0,C 180,E1 -24678.432,E2 -24678.432} C_VEL
LIN {X 0,Y 212.25,Z 381.597,A -85,B 0,C 180,E1 -24678.955,E2 -24678.955} C_VEL
LIN {X 0,Y 209.051,Z 415.726,A -85,B 0,C 180,E1 -24679.897,E2 -24679.897} C_VEL
LIN {X 0,Y 206.532,Z 430.227,A -85,B 0,C 180,E1 -24680.515,E2 -24680.515} C_VEL
LIN {X 0,Y 203.229,Z 443.357,A -85,B 0,C 180,E1 -24681.327,E2 -24681.327} C_VEL
LIN {X 0,Y 198.749,Z 457.001,A -85,B 0,C 180,E1 -24682.514,E2 -24682.514} C_VEL
LIN {X 0,Y 193.594,Z 469.566,A -85,B 0,C 180,E1 -24683.982,E2 -24683.982} C_VEL
LIN {X 0,Y 188.087,Z 480.685,A -85,B 0,C 180,E1 -24685.655,E2 -24685.655} C_VEL
LIN {X 0,Y 181.796,Z 491.549,A -85,B 0,C 180,E1 -24687.764,E2 -24687.764} C_VEL
LIN {X 0,Y 174.964,Z 501.632,A -85,B 0,C 180,E1 -24690.278,E2 -24690.278} C_VEL
LIN {X 0,Y 168.062,Z 510.619,A -85,B 0,C 180,E1 -24693.245,E2 -24693.245} C_VEL
LIN {X 0,Y 160.6,Z 519.117,A -85,B 0,C 180,E1 -24697.002,E2 -24697.002} C_VEL
LIN {X 0,Y 153.896,Z 525.861,A -85,B 0,C 180,E1 -24701.107,E2 -24701.107} C_VEL
LIN {X 0,Y 148.511,Z 530.784,A -85,B 0,C 180,E1 -24705.217,E2 -24705.217} C_VEL
LIN {X 0,Y 143.148,Z 535.078,A -85,B 0,C 180,E1 -24710.34,E2 -24710.34} C_VEL
LIN {X 0,Y 138.712,Z 538.094,A -85,B 0,C 180,E1 -24716.13,E2 -24716.13} C_VEL
LIN {X 0,Y 135.655,Z 539.637,A -85,B 0,C 180,E1 -24722.209,E2 -24722.209} C_VEL
LIN {X 0,Y 133.779,Z 539.763,A -85,B 0,C 180,E1 -24728.425,E2 -24728.425} C_VEL
LIN {X 0,Y 133.374,Z 539.298,A -85,B 0,C 180,E1 -24731.57,E2 -24731.57} C_VEL
LIN {X 0,Y 133.018,Z 537.332,A -85,B 0,C 180,E1 -24737.8,E2 -24737.8} C_VEL
LIN {X 0,Y 133.694,Z 533.918,A -85,B 0,C 180,E1 -24743.966,E2 -24743.966} C_VEL
LIN {X 0,Y 134.728,Z 530.399,A -85,B 0,C 180,E1 -24748.506,E2 -24748.506} C_VEL
LIN {X 0,Y 136.179,Z 525.966,A -85,B 0,C 180,E1 -24752.959,E2 -24752.959} C_VEL
LIN {X 0,Y 138.674,Z 519.554,A -85,B 0,C 180,E1 -24758.012,E2 -24758.012} C_VEL
LIN {X 0,Y 142.107,Z 511.581,A -85,B 0,C 180,E1 -24762.859,E2 -24762.859} C_VEL
LIN {X 0,Y 145.75,Z 503.238,A -85,B 0,C 180,E1 -24766.817,E2 -24766.817} C_VEL
LIN {X 0,Y 150.155,Z 492.827,A -85,B 0,C 180,E1 -24770.694,E2 -24770.694} C_VEL
LIN {X 0,Y 154.089,Z 482.755,A -85,B 0,C 180,E1 -24773.627,E2 -24773.627} C_VEL
LIN {X 0,Y 158.146,Z 470.848,A -85,B 0,C 180,E1 -24776.385,E2 -24776.385} C_VEL
LIN {X 0,Y 161.139,Z 460.435,A -85,B 0,C 180,E1 -24778.314,E2 -24778.314} C_VEL
LIN {X 0,Y 164.667,Z 447.48,A -85,B 0,C 180,E1 -24780.098,E2 -24780.098} C_VEL
LIN {X 0,Y 167.358,Z 433.595,A -85,B 0,C 180,E1 -24781.574,E2 -24781.574} C_VEL
LIN {X 0,Y 169.356,Z 419.965,A -85,B 0,C 180,E1 -24782.559,E2 -24782.559} C_VEL
LIN {X 0,Y 170.829,Z 403.231,A -85,B 0,C 180,E1 -24783.293,E2 -24783.293} C_VEL
LIN {X 0,Y 174.381,Z 351.417,A -85,B 0,C 180,E1 -24785.12,E2 -24785.12} C_VEL
LIN {X 0,Y 168.606,Z 339.157,A -85,B 0,C 180,E1 -24787.735,E2 -24787.735} C_VEL
LIN {X 0,Y 162.872,Z 328.7,A -85,B 0,C 180,E1 -24790.543,E2 -24790.543} C_VEL
LIN {X 0,Y 156.78,Z 318.875,A -85,B 0,C 180,E1 -24793.857,E2 -24793.857} C_VEL
LIN {X 0,Y 151.373,Z 311.145,A -85,B 0,C 180,E1 -24797.168,E2 -24797.168} C_VEL
LIN {X 0,Y 148.563,Z 307.175,A -85,B 0,C 180,E1 -24799.09,E2 -24799.09} C_VEL
LIN {X 0,Y 145.703,Z 303.824,A -85,B 0,C 180,E1 -24801.172,E2 -24801.172} C_VEL
LIN {X 0,Y 144.642,Z 302.109,A -85,B 0,C 180,E1 -24802.045,E2 -24802.045} C_VEL
LIN {X 0,Y 141.981,Z 299.494,A -85,B 0,C 180,E1 -24804.223,E2 -24804.223} C_VEL
LIN {X 0,Y 140.564,Z 296.866,A -85,B 0,C 180,E1 -24805.624,E2 -24805.624} C_VEL
LIN {X 0,Y 137.698,Z 294.854,A -85,B 0,C 180,E1 -24808.354,E2 -24808.354} C_VEL
LIN {X 0,Y 136.332,Z 292.415,A -85,B 0,C 180,E1 -24810.01,E2 -24810.01} C_VEL
LIN {X 0,Y 136.073,Z 291.135,A -85,B 0,C 180,E1 -24810.548,E2 -24810.548} C_VEL
LIN {X 0,Y 136.076,Z 291.134,A -85,B 0,C 180,E1 -24815.6,E2 -24815.6} C_VEL
LIN {X 0,Y 136.238,Z 291.136,A -85,B 0,C 180,E1 -24818.837,E2 -24818.837} C_VEL
LIN {X 0,Y 136.26,Z 291.126,A -85,B 0,C 180,E1 -24825.059,E2 -24825.059} C_VEL
LIN {X 0,Y 136.428,Z 291.116,A -85,B 0,C 180,E1 -24828.17,E2 -24828.17} C_VEL
LIN {X 0,Y 136.538,Z 291.068,A -85,B 0,C 180,E1 -24831.121,E2 -24831.121} C_VEL
LIN {X 0,Y 137.13,Z 291.01,A -85,B 0,C 180,E1 -24840.004,E2 -24840.004} C_VEL
LIN {X 0,Y 136.55,Z 291.095,A -85,B 0,C 180,E1 -24848.886,E2 -24848.886} C_VEL
LIN {X 0,Y 136.418,Z 291.08,A -85,B 0,C 180,E1 -24851.896,E2 -24851.896} C_VEL
LIN {X 0,Y 136.227,Z 291.136,A -85,B 0,C 180,E1 -24855.335,E2 -24855.335} C_VEL
LIN {X 0,Y 136.959,Z 293.515,A -85,B 0,C 180,E1 -24856.397,E2 -24856.397} C_VEL
LIN {X 0,Y 138.851,Z 295.833,A -85,B 0,C 180,E1 -24858.446,E2 -24858.446} C_VEL
LIN {X 0,Y 140.837,Z 297.114,A -85,B 0,C 180,E1 -24860.258,E2 -24860.258} C_VEL
LIN {X 0,Y 142.473,Z 300.168,A -85,B 0,C 180,E1 -24861.846,E2 -24861.846} C_VEL
LIN {X 0,Y 145.094,Z 302.652,A -85,B 0,C 180,E1 -24863.937,E2 -24863.937} C_VEL
LIN {X 0,Y 147.327,Z 305.995,A -85,B 0,C 180,E1 -24865.68,E2 -24865.68} C_VEL
LIN {X 0,Y 148.969,Z 307.795,A -85,B 0,C 180,E1 -24866.823,E2 -24866.823} C_VEL
LIN {X 0,Y 152.611,Z 312.972,A -85,B 0,C 180,E1 -24869.269,E2 -24869.269} C_VEL
LIN {X 0,Y 156.073,Z 318.011,A -85,B 0,C 180,E1 -24871.377,E2 -24871.377} C_VEL
LIN {X 0,Y 161.777,Z 326.974,A -85,B 0,C 180,E1 -24874.519,E2 -24874.519} C_VEL
LIN {X 0,Y 166.995,Z 338.39,A -85,B 0,C 180,E1 -24877.266,E2 -24877.266} C_VEL
LIN {X 0,Y 171.44,Z 349.94,A -85,B 0,C 180,E1 -24879.484,E2 -24879.484} C_VEL
LIN {X 0,Y 174.1,Z 358.028,A -85,B 0,C 180,E1 -24880.786,E2 -24880.786} C_VEL
LIN {X 0,Y 169.745,Z 422.07,A -85,B 0,C 180,E1 -24883.137,E2 -24883.137} C_VEL
LIN {X 0,Y 167.73,Z 436.795,A -85,B 0,C 180,E1 -24884.041,E2 -24884.041} C_VEL
LIN {X 0,Y 165.106,Z 449.668,A -85,B 0,C 180,E1 -24885.171,E2 -24885.171} C_VEL
LIN {X 0,Y 161.853,Z 463.022,A -85,B 0,C 180,E1 -24886.852,E2 -24886.852} C_VEL
LIN {X 0,Y 158.077,Z 475.591,A -85,B 0,C 180,E1 -24888.938,E2 -24888.938} C_VEL
LIN {X 0,Y 154.514,Z 486.415,A -85,B 0,C 180,E1 -24891.288,E2 -24891.288} C_VEL
LIN {X 0,Y 151.491,Z 494.287,A -85,B 0,C 180,E1 -24893.324,E2 -24893.324} C_VEL
LIN {X 0,Y 147.168,Z 504.755,A -85,B 0,C 180,E1 -24896.69,E2 -24896.69} C_VEL
LIN {X 0,Y 143.192,Z 514.201,A -85,B 0,C 180,E1 -24900.607,E2 -24900.607} C_VEL
LIN {X 0,Y 139.766,Z 522.257,A -85,B 0,C 180,E1 -24904.846,E2 -24904.846} C_VEL
LIN {X 0,Y 137.3,Z 528.545,A -85,B 0,C 180,E1 -24909.004,E2 -24909.004} C_VEL
LIN {X 0,Y 136.182,Z 531.635,A -85,B 0,C 180,E1 -24911.435,E2 -24911.435} C_VEL
LIN {X 0,Y 134.709,Z 534.205,A -85,B 0,C 180,E1 -24913.599,E2 -24913.599} C_VEL
LIN {X 0,Y 130.865,Z 537.853,A -85,B 0,C 180,E1 -24917.218,E2 -24917.218} C_VEL
LIN {X 0,Y 127.894,Z 540.26,A -85,B 0,C 180,E1 -24920.326,E2 -24920.326} C_VEL
LIN {X 0,Y 126.558,Z 541.805,A -85,B 0,C 180,E1 -24922.847,E2 -24922.847} C_VEL
LIN {X 0,Y 126.396,Z 542.27,A -85,B 0,C 180,E1 -24923.719,E2 -24923.719} C_VEL
LIN {X 0,Y 126.475,Z 545.156,A -85,B 0,C 180,E1 -24930,E2 -24930} C_VEL
LIN {X 0,Y 126.376,Z 546.079,A -85,B 0,C 180,E1 -24933.188,E2 -24933.188} C_VEL
LIN {X 0,Y 126.713,Z 546.918,A -85,B 0,C 180,E1 -24939.577,E2 -24939.577} C_VEL
LIN {X 0,Y 128.238,Z 546.457,A -85,B 0,C 180,E1 -24945.903,E2 -24945.903} C_VEL
LIN {X 0,Y 131.245,Z 544.706,A -85,B 0,C 180,E1 -24952.014,E2 -24952.014} C_VEL
LIN {X 0,Y 135.547,Z 541.628,A -85,B 0,C 180,E1 -24957.816,E2 -24957.816} C_VEL
LIN {X 0,Y 141.178,Z 537.139,A -85,B 0,C 180,E1 -24963.201,E2 -24963.201} C_VEL
LIN {X 0,Y 148.039,Z 531.085,A -85,B 0,C 180,E1 -24968.108,E2 -24968.108} C_VEL
LIN {X 0,Y 154.886,Z 524.337,A -85,B 0,C 180,E1 -24972.01,E2 -24972.01} C_VEL
LIN {X 0,Y 162.529,Z 515.981,A -85,B 0,C 180,E1 -24975.517,E2 -24975.517} C_VEL
LIN {X 0,Y 169.43,Z 507.314,A -85,B 0,C 180,E1 -24978.299,E2 -24978.299} C_VEL
LIN {X 0,Y 175.46,Z 498.785,A -85,B 0,C 180,E1 -24980.447,E2 -24980.447} C_VEL
LIN {X 0,Y 182.534,Z 487.475,A -85,B 0,C 180,E1 -24982.569,E2 -24982.569} C_VEL
LIN {X 0,Y 188.435,Z 476.285,A -85,B 0,C 180,E1 -24984.211,E2 -24984.211} C_VEL
LIN {X 0,Y 193.933,Z 464.064,A -85,B 0,C 180,E1 -24985.53,E2 -24985.53} C_VEL
LIN {X 0,Y 198.758,Z 450.524,A -85,B 0,C 180,E1 -24986.652,E2 -24986.652} C_VEL
LIN {X 0,Y 202.556,Z 436.639,A -85,B 0,C 180,E1 -24987.465,E2 -24987.465} C_VEL
LIN {X 0,Y 205.125,Z 423.198,A -85,B 0,C 180,E1 -24988.017,E2 -24988.017} C_VEL
LIN {X 0,Y 207.679,Z 398.687,A -85,B 0,C 180,E1 -24988.711,E2 -24988.711} C_VEL
LIN {X 0,Y 208.416,Z 390.014,A -85,B 0,C 180,E1 -24988.981,E2 -24988.981} C_VEL
LIN {X 0,Y 205.088,Z 381.209,A -85,B 0,C 180,E1 -24991.886,E2 -24991.886} C_VEL
LIN {X 0,Y 202.281,Z 374.472,A -85,B 0,C 180,E1 -24994.675,E2 -24994.675} C_VEL
LIN {X 0,Y 200.364,Z 370.274,A -85,B 0,C 180,E1 -24996.835,E2 -24996.835} C_VEL
LIN {X 0,Y 198.429,Z 366.235,A -85,B 0,C 180,E1 -24999.353,E2 -24999.353} C_VEL
LIN {X 0,Y 196.944,Z 363.274,A -85,B 0,C 180,E1 -25001.685,E2 -25001.685} C_VEL
LIN {X 0,Y 194.927,Z 359.894,A -85,B 0,C 180,E1 -25005.912,E2 -25005.912} C_VEL
LIN {X 0,Y 194.642,Z 359.049,A -85,B 0,C 180,E1 -25006.849,E2 -25006.849} C_VEL
LIN {X 0,Y 193.59,Z 358.03,A -85,B 0,C 180,E1 -25011.648,E2 -25011.648} C_VEL
LIN {X 0,Y 194.319,Z 358.402,A -85,B 0,C 180,E1 -25018.443,E2 -25018.443} C_VEL
LIN {X 0,Y 194.855,Z 359.026,A -85,B 0,C 180,E1 -25020.098,E2 -25020.098} C_VEL
LIN {X 0,Y 196.692,Z 362.629,A -85,B 0,C 180,E1 -25024.261,E2 -25024.261} C_VEL
LIN {X 0,Y 197.416,Z 363.94,A -85,B 0,C 180,E1 -25025.495,E2 -25025.495} C_VEL
LIN {X 0,Y 199.785,Z 368.047,A -85,B 0,C 180,E1 -25028.755,E2 -25028.755} C_VEL
LIN {X 0,Y 202.471,Z 372.842,A -85,B 0,C 180,E1 -25031.732,E2 -25031.732} C_VEL
LIN {X 0,Y 205.881,Z 379.19,A -85,B 0,C 180,E1 -25034.899,E2 -25034.899} C_VEL
LIN {X 0,Y 208.846,Z 385.191,A -85,B 0,C 180,E1 -25037.307,E2 -25037.307} C_VEL
LIN {X 0,Y 205.665,Z 417.213,A -85,B 0,C 180,E1 -25038.201,E2 -25038.201} C_VEL
LIN {X 0,Y 203.002,Z 431.539,A -85,B 0,C 180,E1 -25038.813,E2 -25038.813} C_VEL
LIN {X 0,Y 199.583,Z 444.481,A -85,B 0,C 180,E1 -25039.621,E2 -25039.621} C_VEL
LIN {X 0,Y 194.898,Z 458.129,A -85,B 0,C 180,E1 -25040.811,E2 -25040.811} C_VEL
LIN {X 0,Y 189.762,Z 470.113,A -85,B 0,C 180,E1 -25042.2,E2 -25042.2} C_VEL
LIN {X 0,Y 183.655,Z 481.967,A -85,B 0,C 180,E1 -25043.991,E2 -25043.991} C_VEL
LIN {X 0,Y 176.906,Z 493.034,A -85,B 0,C 180,E1 -25046.17,E2 -25046.17} C_VEL
LIN {X 0,Y 170.09,Z 502.578,A -85,B 0,C 180,E1 -25048.597,E2 -25048.597} C_VEL
LIN {X 0,Y 162.927,Z 511.428,A -85,B 0,C 180,E1 -25051.58,E2 -25051.58} C_VEL
LIN {X 0,Y 156.227,Z 518.721,A -85,B 0,C 180,E1 -25054.818,E2 -25054.818} C_VEL
LIN {X 0,Y 149.076,Z 525.597,A -85,B 0,C 180,E1 -25058.936,E2 -25058.936} C_VEL
LIN {X 0,Y 142.617,Z 531.125,A -85,B 0,C 180,E1 -25063.616,E2 -25063.616} C_VEL
LIN {X 0,Y 137.462,Z 535.026,A -85,B 0,C 180,E1 -25068.346,E2 -25068.346} C_VEL
LIN {X 0,Y 132.573,Z 538.138,A -85,B 0,C 180,E1 -25074.33,E2 -25074.33} C_VEL
LIN {X 0,Y 129.101,Z 539.776,A -85,B 0,C 180,E1 -25080.664,E2 -25080.664} C_VEL
LIN {X 0,Y 126.925,Z 539.994,A -85,B 0,C 180,E1 -25087.196,E2 -25087.196} C_VEL
LIN {X 0,Y 126.296,Z 539.486,A -85,B 0,C 180,E1 -25091.069,E2 -25091.069} C_VEL
LIN {X 0,Y 125.901,Z 537.705,A -85,B 0,C 180,E1 -25097.099,E2 -25097.099} C_VEL
LIN {X 0,Y 126.519,Z 534.417,A -85,B 0,C 180,E1 -25103.622,E2 -25103.622} C_VEL
LIN {X 0,Y 127.587,Z 530.946,A -85,B 0,C 180,E1 -25108.422,E2 -25108.422} C_VEL
LIN {X 0,Y 129.058,Z 526.616,A -85,B 0,C 180,E1 -25113.122,E2 -25113.122} C_VEL
LIN {X 0,Y 131.621,Z 520.315,A -85,B 0,C 180,E1 -25118.444,E2 -25118.444} C_VEL
LIN {X 0,Y 135.161,Z 512.468,A -85,B 0,C 180,E1 -25123.532,E2 -25123.532} C_VEL
LIN {X 0,Y 138.959,Z 504.263,A -85,B 0,C 180,E1 -25127.665,E2 -25127.665} C_VEL
LIN {X 0,Y 143.538,Z 494.016,A -85,B 0,C 180,E1 -25131.695,E2 -25131.695} C_VEL
LIN {X 0,Y 147.689,Z 483.926,A -85,B 0,C 180,E1 -25134.794,E2 -25134.794} C_VEL
LIN {X 0,Y 151.817,Z 472.517,A -85,B 0,C 180,E1 -25137.576,E2 -25137.576} C_VEL
LIN {X 0,Y 154.92,Z 462.391,A -85,B 0,C 180,E1 -25139.56,E2 -25139.56} C_VEL
LIN {X 0,Y 158.624,Z 449.862,A -85,B 0,C 180,E1 -25141.372,E2 -25141.372} C_VEL
LIN {X 0,Y 161.527,Z 436.123,A -85,B 0,C 180,E1 -25142.947,E2 -25142.947} C_VEL
LIN {X 0,Y 163.823,Z 421.758,A -85,B 0,C 180,E1 -25144.078,E2 -25144.078} C_VEL
LIN {X 0,Y 165.336,Z 406.365,A -85,B 0,C 180,E1 -25144.808,E2 -25144.808} C_VEL
LIN {X 0,Y 169.166,Z 353.88,A -85,B 0,C 180,E1 -25146.657,E2 -25146.657} C_VEL
LIN {X 0,Y 163.552,Z 341.915,A -85,B 0,C 180,E1 -25149.411,E2 -25149.411} C_VEL
LIN {X 0,Y 158.349,Z 332.372,A -85,B 0,C 180,E1 -25152.178,E2 -25152.178} C_VEL
LIN {X 0,Y 153.112,Z 323.855,A -85,B 0,C 180,E1 -25155.246,E2 -25155.246} C_VEL
LIN {X 0,Y 148.585,Z 317.075,A -85,B 0,C 180,E1 -25158.217,E2 -25158.217} C_VEL
LIN {X 0,Y 145.315,Z 312.617,A -85,B 0,C 180,E1 -25160.593,E2 -25160.593} C_VEL
LIN {X 0,Y 142.681,Z 308.985,A -85,B 0,C 180,E1 -25162.72,E2 -25162.72} C_VEL
LIN {X 0,Y 139.175,Z 304.797,A -85,B 0,C 180,E1 -25165.856,E2 -25165.856} C_VEL
LIN {X 0,Y 138.453,Z 303.437,A -85,B 0,C 180,E1 -25166.624,E2 -25166.624} C_VEL
LIN {X 0,Y 135.624,Z 301.031,A -85,B 0,C 180,E1 -25169.55,E2 -25169.55} C_VEL
LIN {X 0,Y 134.151,Z 298.183,A -85,B 0,C 180,E1 -25171.516,E2 -25171.516} C_VEL
LIN {X 0,Y 130.638,Z 295.695,A -85,B 0,C 180,E1 -25176.477,E2 -25176.477} C_VEL
LIN {X 0,Y 129.459,Z 293.267,A -85,B 0,C 180,E1 -25178.964,E2 -25178.964} C_VEL
LIN {X 0,Y 129.149,Z 292.013,A -85,B 0,C 180,E1 -25179.914,E2 -25179.914} C_VEL
LIN {X 0,Y 129.186,Z 292.011,A -85,B 0,C 180,E1 -25184.221,E2 -25184.221} C_VEL
LIN {X 0,Y 129.386,Z 291.993,A -85,B 0,C 180,E1 -25187.881,E2 -25187.881} C_VEL
LIN {X 0,Y 129.463,Z 291.952,A -85,B 0,C 180,E1 -25190.632,E2 -25190.632} C_VEL
LIN {X 0,Y 130.085,Z 291.885,A -85,B 0,C 180,E1 -25200.004,E2 -25200.004} C_VEL
LIN {X 0,Y 129.493,Z 292.049,A -85,B 0,C 180,E1 -25206.431,E2 -25206.431} C_VEL
LIN {X 0,Y 130.095,Z 294.137,A -85,B 0,C 180,E1 -25207.961,E2 -25207.961} C_VEL
LIN {X 0,Y 132,Z 296.636,A -85,B 0,C 180,E1 -25211.25,E2 -25211.25} C_VEL
LIN {X 0,Y 134.316,Z 298.201,A -85,B 0,C 180,E1 -25214.298,E2 -25214.298} C_VEL
LIN {X 0,Y 135.867,Z 301.15,A -85,B 0,C 180,E1 -25216.34,E2 -25216.34} C_VEL
LIN {X 0,Y 138.342,Z 303.307,A -85,B 0,C 180,E1 -25218.9,E2 -25218.9} C_VEL
LIN {X 0,Y 141.067,Z 307.383,A -85,B 0,C 180,E1 -25221.56,E2 -25221.56} C_VEL
LIN {X 0,Y 142.757,Z 309.069,A -85,B 0,C 180,E1 -25222.968,E2 -25222.968} C_VEL
LIN {X 0,Y 145.375,Z 312.699,A -85,B 0,C 180,E1 -25225.076,E2 -25225.076} C_VEL
LIN {X 0,Y 149.236,Z 318.069,A -85,B 0,C 180,E1 -25227.86,E2 -25227.86} C_VEL
LIN {X 0,Y 154.185,Z 325.589,A -85,B 0,C 180,E1 -25231.044,E2 -25231.044} C_VEL
LIN {X 0,Y 158.652,Z 333.109,A -85,B 0,C 180,E1 -25233.627,E2 -25233.627} C_VEL
LIN {X 0,Y 164.055,Z 346.004,A -85,B 0,C 180,E1 -25236.664,E2 -25236.664} C_VEL
LIN {X 0,Y 168.008,Z 357.208,A -85,B 0,C 180,E1 -25238.771,E2 -25238.771} C_VEL
LIN {X 0,Y 168.81,Z 359.827,A -85,B 0,C 180,E1 -25239.198,E2 -25239.198} C_VEL
LIN {X 0,Y 164.822,Z 417.678,A -85,B 0,C 180,E1 -25241.344,E2 -25241.344} C_VEL
LIN {X 0,Y 163.085,Z 432.142,A -85,B 0,C 180,E1 -25242.12,E2 -25242.12} C_VEL
LIN {X 0,Y 160.743,Z 444.893,A -85,B 0,C 180,E1 -25243.147,E2 -25243.147} C_VEL
LIN {X 0,Y 157.761,Z 457.39,A -85,B 0,C 180,E1 -25244.54,E2 -25244.54} C_VEL
LIN {X 0,Y 154.076,Z 469.833,A -85,B 0,C 180,E1 -25246.378,E2 -25246.378} C_VEL
LIN {X 0,Y 150.364,Z 481.394,A -85,B 0,C 180,E1 -25248.686,E2 -25248.686} C_VEL
LIN {X 0,Y 145.761,Z 493.153,A -85,B 0,C 180,E1 -25251.628,E2 -25251.628} C_VEL
LIN {X 0,Y 141.242,Z 503.795,A -85,B 0,C 180,E1 -25255.095,E2 -25255.095} C_VEL
LIN {X 0,Y 136.967,Z 513.391,A -85,B 0,C 180,E1 -25259.129,E2 -25259.129} C_VEL
LIN {X 0,Y 133.056,Z 522.132,A -85,B 0,C 180,E1 -25263.895,E2 -25263.895} C_VEL
LIN {X 0,Y 129.875,Z 529.839,A -85,B 0,C 180,E1 -25269.406,E2 -25269.406} C_VEL
LIN {X 0,Y 127.974,Z 534.95,A -85,B 0,C 180,E1 -25274.063,E2 -25274.063} C_VEL
LIN {X 0,Y 126.71,Z 540.194,A -85,B 0,C 180,E1 -25280.422,E2 -25280.422} C_VEL
LIN {X 0,Y 126.396,Z 542.27,A -85,B 0,C 180,E1 -25283.719,E2 -25283.719} C_VEL
LIN {X 0,Y 125.554,Z 543.622,A -85,B 0,C 180,E1 -25286.317,E2 -25286.317} C_VEL
LIN {X 0,Y 123.885,Z 544.664,A -85,B 0,C 180,E1 -25288.9,E2 -25288.9} C_VEL
LIN {X 0,Y 120.257,Z 546.037,A -85,B 0,C 180,E1 -25294.251,E2 -25294.251} C_VEL
LIN {X 0,Y 119.407,Z 546.455,A -85,B 0,C 180,E1 -25297.09,E2 -25297.09} C_VEL
LIN {X 0,Y 119.411,Z 546.52,A -85,B 0,C 180,E1 -25298.051,E2 -25298.051} C_VEL
LIN {X 0,Y 120.403,Z 546.666,A -85,B 0,C 180,E1 -25303.501,E2 -25303.501} C_VEL
LIN {X 0,Y 122.806,Z 545.628,A -85,B 0,C 180,E1 -25310.081,E2 -25310.081} C_VEL
LIN {X 0,Y 126.792,Z 543.291,A -85,B 0,C 180,E1 -25316.322,E2 -25316.322} C_VEL
LIN {X 0,Y 132.071,Z 539.594,A -85,B 0,C 180,E1 -25322.149,E2 -25322.149} C_VEL
LIN {X 0,Y 138.744,Z 534.433,A -85,B 0,C 180,E1 -25327.433,E2 -25327.433} C_VEL
LIN {X 0,Y 144.492,Z 529.466,A -85,B 0,C 180,E1 -25331.042,E2 -25331.042} C_VEL
LIN {X 0,Y 151.924,Z 522.387,A -85,B 0,C 180,E1 -25334.865,E2 -25334.865} C_VEL
LIN {X 0,Y 159.996,Z 513.664,A -85,B 0,C 180,E1 -25338.307,E2 -25338.307} C_VEL
LIN {X 0,Y 166.997,Z 504.903,A -85,B 0,C 180,E1 -25340.935,E2 -25340.935} C_VEL
LIN {X 0,Y 173.677,Z 495.544,A -85,B 0,C 180,E1 -25343.052,E2 -25343.052} C_VEL
LIN {X 0,Y 181.034,Z 483.638,A -85,B 0,C 180,E1 -25345.093,E2 -25345.093} C_VEL
LIN {X 0,Y 187.181,Z 471.682,A -85,B 0,C 180,E1 -25346.656,E2 -25346.656} C_VEL
LIN {X 0,Y 192.148,Z 460.183,A -85,B 0,C 180,E1 -25347.757,E2 -25347.757} C_VEL
LIN {X 0,Y 196.762,Z 446.741,A -85,B 0,C 180,E1 -25348.758,E2 -25348.758} C_VEL
LIN {X 0,Y 200.456,Z 432.26,A -85,B 0,C 180,E1 -25349.5,E2 -25349.5} C_VEL
LIN {X 0,Y 202.88,Z 417.766,A -85,B 0,C 180,E1 -25349.998,E2 -25349.998} C_VEL
LIN {X 0,Y 205.234,Z 393.33,A -85,B 0,C 180,E1 -25350.685,E2 -25350.685} C_VEL
LIN {X 0,Y 201.922,Z 384.292,A -85,B 0,C 180,E1 -25353.922,E2 -25353.922} C_VEL
LIN {X 0,Y 199.109,Z 377.374,A -85,B 0,C 180,E1 -25357.15,E2 -25357.15} C_VEL
LIN {X 0,Y 196.928,Z 372.621,A -85,B 0,C 180,E1 -25360.144,E2 -25360.144} C_VEL
LIN {X 0,Y 195.657,Z 369.983,A -85,B 0,C 180,E1 -25362.313,E2 -25362.313} C_VEL
LIN {X 0,Y 193.831,Z 366.619,A -85,B 0,C 180,E1 -25366.499,E2 -25366.499} C_VEL
LIN {X 0,Y 193.563,Z 365.971,A -85,B 0,C 180,E1 -25367.414,E2 -25367.414} C_VEL
LIN {X 0,Y 192.714,Z 365.09,A -85,B 0,C 180,E1 -25371.609,E2 -25371.609} C_VEL
LIN {X 0,Y 193.289,Z 365.337,A -85,B 0,C 180,E1 -25377.913,E2 -25377.913} C_VEL
LIN {X 0,Y 193.834,Z 365.981,A -85,B 0,C 180,E1 -25379.738,E2 -25379.738} C_VEL
LIN {X 0,Y 195.701,Z 369.662,A -85,B 0,C 180,E1 -25384.116,E2 -25384.116} C_VEL
LIN {X 0,Y 198.272,Z 374.573,A -85,B 0,C 180,E1 -25388.073,E2 -25388.073} C_VEL
LIN {X 0,Y 200.796,Z 379.294,A -85,B 0,C 180,E1 -25391.04,E2 -25391.04} C_VEL
LIN {X 0,Y 204.161,Z 385.88,A -85,B 0,C 180,E1 -25394.33,E2 -25394.33} C_VEL
LIN {X 0,Y 205.618,Z 388.997,A -85,B 0,C 180,E1 -25395.609,E2 -25395.609} C_VEL
LIN {X 0,Y 202.703,Z 417.313,A -85,B 0,C 180,E1 -25396.393,E2 -25396.393} C_VEL
LIN {X 0,Y 199.976,Z 431.671,A -85,B 0,C 180,E1 -25396.991,E2 -25396.991} C_VEL
LIN {X 0,Y 196.481,Z 444.534,A -85,B 0,C 180,E1 -25397.762,E2 -25397.762} C_VEL
LIN {X 0,Y 191.732,Z 458.043,A -85,B 0,C 180,E1 -25398.912,E2 -25398.912} C_VEL
LIN {X 0,Y 186.38,Z 470.201,A -85,B 0,C 180,E1 -25400.288,E2 -25400.288} C_VEL
LIN {X 0,Y 180.067,Z 482.054,A -85,B 0,C 180,E1 -25402.038,E2 -25402.038} C_VEL
LIN {X 0,Y 173.73,Z 492.172,A -85,B 0,C 180,E1 -25403.989,E2 -25403.989} C_VEL
LIN {X 0,Y 166.646,Z 501.834,A -85,B 0,C 180,E1 -25406.343,E2 -25406.343} C_VEL
LIN {X 0,Y 159.483,Z 510.456,A -85,B 0,C 180,E1 -25409.14,E2 -25409.14} C_VEL
LIN {X 0,Y 152.06,Z 518.276,A -85,B 0,C 180,E1 -25412.492,E2 -25412.492} C_VEL
LIN {X 0,Y 144.47,Z 525.311,A -85,B 0,C 180,E1 -25416.616,E2 -25416.616} C_VEL
LIN {X 0,Y 138.652,Z 530.086,A -85,B 0,C 180,E1 -25420.51,E2 -25420.51} C_VEL
LIN {X 0,Y 131.943,Z 534.963,A -85,B 0,C 180,E1 -25426.177,E2 -25426.177} C_VEL
LIN {X 0,Y 126.563,Z 538.183,A -85,B 0,C 180,E1 -25432.352,E2 -25432.352} C_VEL
LIN {X 0,Y 122.642,Z 539.915,A -85,B 0,C 180,E1 -25438.954,E2 -25438.954} C_VEL
LIN {X 0,Y 120.115,Z 540.225,A -85,B 0,C 180,E1 -25445.823,E2 -25445.823} C_VEL
LIN {X 0,Y 119.273,Z 539.673,A -85,B 0,C 180,E1 -25450.507,E2 -25450.507} C_VEL
LIN {X 0,Y 118.801,Z 538.069,A -85,B 0,C 180,E1 -25456.313,E2 -25456.313} C_VEL
LIN {X 0,Y 119.32,Z 534.885,A -85,B 0,C 180,E1 -25463.235,E2 -25463.235} C_VEL
LIN {X 0,Y 120.437,Z 531.494,A -85,B 0,C 180,E1 -25468.328,E2 -25468.328} C_VEL
LIN {X 0,Y 122.586,Z 525.64,A -85,B 0,C 180,E1 -25474.934,E2 -25474.934} C_VEL
LIN {X 0,Y 125.558,Z 519.045,A -85,B 0,C 180,E1 -25480.481,E2 -25480.481} C_VEL
LIN {X 0,Y 129.527,Z 510.859,A -85,B 0,C 180,E1 -25485.741,E2 -25485.741} C_VEL
LIN {X 0,Y 133.669,Z 502.288,A -85,B 0,C 180,E1 -25489.984,E2 -25489.984} C_VEL
LIN {X 0,Y 138.462,Z 491.894,A -85,B 0,C 180,E1 -25493.958,E2 -25493.958} C_VEL
LIN {X 0,Y 142.847,Z 481.458,A -85,B 0,C 180,E1 -25497.071,E2 -25497.071} C_VEL
LIN {X 0,Y 146.965,Z 470.148,A -85,B 0,C 180,E1 -25499.745,E2 -25499.745} C_VEL
LIN {X 0,Y 150.337,Z 459.558,A -85,B 0,C 180,E1 -25501.73,E2 -25501.73} C_VEL
LIN {X 0,Y 153.902,Z 447.279,A -85,B 0,C 180,E1 -25503.424,E2 -25503.424} C_VEL
LIN {X 0,Y 156.82,Z 433.143,A -85,B 0,C 180,E1 -25504.945,E2 -25504.945} C_VEL
LIN {X 0,Y 159.035,Z 418.641,A -85,B 0,C 180,E1 -25505.978,E2 -25505.978} C_VEL
LIN {X 0,Y 160.767,Z 398.615,A -85,B 0,C 180,E1 -25506.826,E2 -25506.826} C_VEL
LIN {X 0,Y 164.018,Z 356.367,A -85,B 0,C 180,E1 -25508.312,E2 -25508.312} C_VEL
LIN {X 0,Y 159.602,Z 346.612,A -85,B 0,C 180,E1 -25510.663,E2 -25510.663} C_VEL
LIN {X 0,Y 154.056,Z 336.209,A -85,B 0,C 180,E1 -25513.846,E2 -25513.846} C_VEL
LIN {X 0,Y 148.282,Z 326.646,A -85,B 0,C 180,E1 -25517.571,E2 -25517.571} C_VEL
LIN {X 0,Y 144.458,Z 321.154,A -85,B 0,C 180,E1 -25520.341,E2 -25520.341} C_VEL
LIN {X 0,Y 142.595,Z 318.477,A -85,B 0,C 180,E1 -25521.828,E2 -25521.828} C_VEL
LIN {X 0,Y 139.738,Z 314.493,A -85,B 0,C 180,E1 -25524.317,E2 -25524.317} C_VEL
LIN {X 0,Y 136.863,Z 310.769,A -85,B 0,C 180,E1 -25527.129,E2 -25527.129} C_VEL
LIN {X 0,Y 136.312,Z 309.844,A -85,B 0,C 180,E1 -25527.74,E2 -25527.74} C_VEL
LIN {X 0,Y 133.728,Z 307.384,A -85,B 0,C 180,E1 -25530.63,E2 -25530.63} C_VEL
LIN {X 0,Y 132.191,Z 304.616,A -85,B 0,C 180,E1 -25532.802,E2 -25532.802} C_VEL
LIN {X 0,Y 129.48,Z 302.69,A -85,B 0,C 180,E1 -25536.868,E2 -25536.868} C_VEL
LIN {X 0,Y 128.17,Z 300.208,A -85,B 0,C 180,E1 -25539.716,E2 -25539.716} C_VEL
LIN {X 0,Y 127.819,Z 299.011,A -85,B 0,C 180,E1 -25540.742,E2 -25540.742} C_VEL
LIN {X 0,Y 125.323,Z 297.734,A -85,B 0,C 180,E1 -25550.319,E2 -25550.319} C_VEL
LIN {X 0,Y 126.274,Z 297.938,A -85,B 0,C 180,E1 -25560.442,E2 -25560.442} C_VEL
LIN {X 0,Y 128.119,Z 299.058,A -85,B 0,C 180,E1 -25565.513,E2 -25565.513} C_VEL
LIN {X 0,Y 129.26,Z 301.778,A -85,B 0,C 180,E1 -25568.21,E2 -25568.21} C_VEL
LIN {X 0,Y 131.461,Z 304.084,A -85,B 0,C 180,E1 -25571.824,E2 -25571.824} C_VEL
LIN {X 0,Y 132.584,Z 304.937,A -85,B 0,C 180,E1 -25573.34,E2 -25573.34} C_VEL
LIN {X 0,Y 134.465,Z 308.161,A -85,B 0,C 180,E1 -25575.882,E2 -25575.882} C_VEL
LIN {X 0,Y 136.624,Z 310.217,A -85,B 0,C 180,E1 -25578.224,E2 -25578.224} C_VEL
LIN {X 0,Y 138.934,Z 313.734,A -85,B 0,C 180,E1 -25580.597,E2 -25580.597} C_VEL
LIN {X 0,Y 140.501,Z 315.506,A -85,B 0,C 180,E1 -25581.998,E2 -25581.998} C_VEL
LIN {X 0,Y 144.427,Z 321.041,A -85,B 0,C 180,E1 -25585.252,E2 -25585.252} C_VEL
LIN {X 0,Y 148.678,Z 327.379,A -85,B 0,C 180,E1 -25588.334,E2 -25588.334} C_VEL
LIN {X 0,Y 154.434,Z 336.954,A -85,B 0,C 180,E1 -25592.016,E2 -25592.016} C_VEL
LIN {X 0,Y 159.108,Z 348.26,A -85,B 0,C 180,E1 -25594.868,E2 -25594.868} C_VEL
LIN {X 0,Y 163.01,Z 359.421,A -85,B 0,C 180,E1 -25597.131,E2 -25597.131} C_VEL
LIN {X 0,Y 163.696,Z 361.718,A -85,B 0,C 180,E1 -25597.53,E2 -25597.53} C_VEL
LIN {X 0,Y 159.288,Z 421.627,A -85,B 0,C 180,E1 -25599.803,E2 -25599.803} C_VEL
LIN {X 0,Y 157.214,Z 435.745,A -85,B 0,C 180,E1 -25600.664,E2 -25600.664} C_VEL
LIN {X 0,Y 154.741,Z 447.655,A -85,B 0,C 180,E1 -25601.708,E2 -25601.708} C_VEL
LIN {X 0,Y 151.177,Z 461.363,A -85,B 0,C 180,E1 -25603.417,E2 -25603.417} C_VEL
LIN {X 0,Y 147.116,Z 473.916,A -85,B 0,C 180,E1 -25605.503,E2 -25605.503} C_VEL
LIN {X 0,Y 142.641,Z 486.368,A -85,B 0,C 180,E1 -25608.307,E2 -25608.307} C_VEL
LIN {X 0,Y 139.322,Z 494.202,A -85,B 0,C 180,E1 -25610.443,E2 -25610.443} C_VEL
LIN {X 0,Y 134.596,Z 504.608,A -85,B 0,C 180,E1 -25614.026,E2 -25614.026} C_VEL
LIN {X 0,Y 130.176,Z 514.004,A -85,B 0,C 180,E1 -25618.239,E2 -25618.239} C_VEL
LIN {X 0,Y 126.353,Z 522.054,A -85,B 0,C 180,E1 -25622.875,E2 -25622.875} C_VEL
LIN {X 0,Y 123.2,Z 529.247,A -85,B 0,C 180,E1 -25628.235,E2 -25628.235} C_VEL
LIN {X 0,Y 121.105,Z 534.427,A -85,B 0,C 180,E1 -25633.132,E2 -25633.132} C_VEL
LIN {X 0,Y 119.926,Z 538.57,A -85,B 0,C 180,E1 -25638.164,E2 -25638.164} C_VEL
LIN {X 0,Y 119.288,Z 542.022,A -85,B 0,C 180,E1 -25643.631,E2 -25643.631} C_VEL
LIN {X 0,Y 119.398,Z 544.837,A -85,B 0,C 180,E1 -25650,E2 -25650} C_VEL
LIN {X 0,Y 119.283,Z 545.793,A -85,B 0,C 180,E1 -25653.377,E2 -25653.377} C_VEL
LIN {X 0,Y 119.411,Z 546.52,A -85,B 0,C 180,E1 -25658.051,E2 -25658.051} C_VEL
LIN {X 0,Y 119.124,Z 546.715,A -85,B 0,C 180,E1 -25660.883,E2 -25660.883} C_VEL
LIN {X 0,Y 117.396,Z 546.473,A -85,B 0,C 180,E1 -25665.614,E2 -25665.614} C_VEL
LIN {X 0,Y 116.42,Z 545.91,A -85,B 0,C 180,E1 -25669.479,E2 -25669.479} C_VEL
LIN {X 0,Y 116.817,Z 545.244,A -85,B 0,C 180,E1 -25672.367,E2 -25672.367} C_VEL
LIN {X 0,Y 117.278,Z 544.931,A -85,B 0,C 180,E1 -25673.299,E2 -25673.299} C_VEL
LIN {X 0,Y 120.439,Z 543.246,A -85,B 0,C 180,E1 -25677.827,E2 -25677.827} C_VEL
LIN {X 0,Y 126.091,Z 539.621,A -85,B 0,C 180,E1 -25683.873,E2 -25683.873} C_VEL
LIN {X 0,Y 133.162,Z 534.537,A -85,B 0,C 180,E1 -25689.295,E2 -25689.295} C_VEL
LIN {X 0,Y 141.312,Z 527.842,A -85,B 0,C 180,E1 -25694.127,E2 -25694.127} C_VEL
LIN {X 0,Y 149.321,Z 520.422,A -85,B 0,C 180,E1 -25697.84,E2 -25697.84} C_VEL
LIN {X 0,Y 157.606,Z 511.586,A -85,B 0,C 180,E1 -25701.063,E2 -25701.063} C_VEL
LIN {X 0,Y 165.48,Z 501.735,A -85,B 0,C 180,E1 -25703.796,E2 -25703.796} C_VEL
LIN {X 0,Y 173.641,Z 490.121,A -85,B 0,C 180,E1 -25706.068,E2 -25706.068} C_VEL
LIN {X 0,Y 180.568,Z 478.286,A -85,B 0,C 180,E1 -25707.835,E2 -25707.835} C_VEL
LIN {X 0,Y 186.324,Z 466.653,A -85,B 0,C 180,E1 -25709.102,E2 -25709.102} C_VEL
LIN {X 0,Y 191.755,Z 453.019,A -85,B 0,C 180,E1 -25710.244,E2 -25710.244} C_VEL
LIN {X 0,Y 196.123,Z 438.574,A -85,B 0,C 180,E1 -25711.088,E2 -25711.088} C_VEL
LIN {X 0,Y 199.124,Z 424.545,A -85,B 0,C 180,E1 -25711.646,E2 -25711.646} C_VEL
LIN {X 0,Y 201.381,Z 405.908,A -85,B 0,C 180,E1 -25712.165,E2 -25712.165} C_VEL
LIN {X 0,Y 202.189,Z 396.728,A -85,B 0,C 180,E1 -25712.469,E2 -25712.469} C_VEL
LIN {X 0,Y 199.685,Z 389.573,A -85,B 0,C 180,E1 -25715.182,E2 -25715.182} C_VEL
LIN {X 0,Y 197.42,Z 383.583,A -85,B 0,C 180,E1 -25718.03,E2 -25718.03} C_VEL
LIN {X 0,Y 195.218,Z 378.369,A -85,B 0,C 180,E1 -25721.411,E2 -25721.411} C_VEL
LIN {X 0,Y 194.441,Z 376.764,A -85,B 0,C 180,E1 -25722.86,E2 -25722.86} C_VEL
LIN {X 0,Y 192.737,Z 373.262,A -85,B 0,C 180,E1 -25727.172,E2 -25727.172} C_VEL
LIN {X 0,Y 191.838,Z 372.144,A -85,B 0,C 180,E1 -25731.571,E2 -25731.571} C_VEL
LIN {X 0,Y 192.404,Z 372.39,A -85,B 0,C 180,E1 -25737.904,E2 -25737.904} C_VEL
LIN {X 0,Y 192.813,Z 372.911,A -85,B 0,C 180,E1 -25739.345,E2 -25739.345} C_VEL
LIN {X 0,Y 194.83,Z 377.201,A -85,B 0,C 180,E1 -25744.245,E2 -25744.245} C_VEL
LIN {X 0,Y 197.007,Z 381.543,A -85,B 0,C 180,E1 -25747.685,E2 -25747.685} C_VEL
LIN {X 0,Y 199.493,Z 386.372,A -85,B 0,C 180,E1 -25750.715,E2 -25750.715} C_VEL
LIN {X 0,Y 202.575,Z 392.948,A -85,B 0,C 180,E1 -25753.872,E2 -25753.872} C_VEL
LIN {X 0,Y 199.925,Z 417.562,A -85,B 0,C 180,E1 -25754.538,E2 -25754.538} C_VEL
LIN {X 0,Y 197.208,Z 431.589,A -85,B 0,C 180,E1 -25755.103,E2 -25755.103} C_VEL
LIN {X 0,Y 193.599,Z 444.596,A -85,B 0,C 180,E1 -25755.852,E2 -25755.852} C_VEL
LIN {X 0,Y 189.24,Z 456.839,A -85,B 0,C 180,E1 -25756.842,E2 -25756.842} C_VEL
LIN {X 0,Y 183.94,Z 468.829,A -85,B 0,C 180,E1 -25758.121,E2 -25758.121} C_VEL
LIN {X 0,Y 177.416,Z 480.961,A -85,B 0,C 180,E1 -25759.816,E2 -25759.816} C_VEL
LIN {X 0,Y 169.978,Z 492.57,A -85,B 0,C 180,E1 -25761.982,E2 -25761.982} C_VEL
LIN {X 0,Y 162.146,Z 502.821,A -85,B 0,C 180,E1 -25764.469,E2 -25764.469} C_VEL
LIN {X 0,Y 153.821,Z 512.245,A -85,B 0,C 180,E1 -25767.618,E2 -25767.618} C_VEL
LIN {X 0,Y 145.813,Z 520.063,A -85,B 0,C 180,E1 -25771.186,E2 -25771.186} C_VEL
LIN {X 0,Y 137.975,Z 526.732,A -85,B 0,C 180,E1 -25775.416,E2 -25775.416} C_VEL
LIN {X 0,Y 131.262,Z 531.78,A -85,B 0,C 180,E1 -25779.973,E2 -25779.973} C_VEL
LIN {X 0,Y 126.625,Z 534.863,A -85,B 0,C 180,E1 -25783.821,E2 -25783.821} C_VEL
LIN {X 0,Y 120.707,Z 538.226,A -85,B 0,C 180,E1 -25790.176,E2 -25790.176} C_VEL
LIN {X 0,Y 116.289,Z 540.054,A -85,B 0,C 180,E1 -25797.05,E2 -25797.05} C_VEL
LIN {X 0,Y 113.371,Z 540.457,A -85,B 0,C 180,E1 -25804.283,E2 -25804.283} C_VEL
LIN {X 0,Y 112.016,Z 539.453,A -85,B 0,C 180,E1 -25811.718,E2 -25811.718} C_VEL
LIN {X 0,Y 111.77,Z 537.065,A -85,B 0,C 180,E1 -25819.127,E2 -25819.127} C_VEL
LIN {X 0,Y 112.835,Z 533.248,A -85,B 0,C 180,E1 -25826.429,E2 -25826.429} C_VEL
LIN {X 0,Y 114.196,Z 529.373,A -85,B 0,C 180,E1 -25831.764,E2 -25831.764} C_VEL
LIN {X 0,Y 116.204,Z 524.602,A -85,B 0,C 180,E1 -25836.948,E2 -25836.948} C_VEL
LIN {X 0,Y 119.636,Z 517.678,A -85,B 0,C 180,E1 -25842.726,E2 -25842.726} C_VEL
LIN {X 0,Y 123.362,Z 510.456,A -85,B 0,C 180,E1 -25847.403,E2 -25847.403} C_VEL
LIN {X 0,Y 127.81,Z 501.76,A -85,B 0,C 180,E1 -25851.788,E2 -25851.788} C_VEL
LIN {X 0,Y 132.542,Z 491.965,A -85,B 0,C 180,E1 -25855.621,E2 -25855.621} C_VEL
LIN {X 0,Y 137.511,Z 480.613,A -85,B 0,C 180,E1 -25859.047,E2 -25859.047} C_VEL
LIN {X 0,Y 141.808,Z 469.095,A -85,B 0,C 180,E1 -25861.774,E2 -25861.774} C_VEL
LIN {X 0,Y 145.437,Z 458.182,A -85,B 0,C 180,E1 -25863.76,E2 -25863.76} C_VEL
LIN {X 0,Y 148.845,Z 446.611,A -85,B 0,C 180,E1 -25865.338,E2 -25865.338} C_VEL
LIN {X 0,Y 151.778,Z 432.916,A -85,B 0,C 180,E1 -25866.802,E2 -25866.802} C_VEL
LIN {X 0,Y 154.062,Z 418.287,A -85,B 0,C 180,E1 -25867.842,E2 -25867.842} C_VEL
LIN {X 0,Y 155.959,Z 397.272,A -85,B 0,C 180,E1 -25868.706,E2 -25868.706} C_VEL
LIN {X 0,Y 159.015,Z 359.43,A -85,B 0,C 180,E1 -25870.034,E2 -25870.034} C_VEL
LIN {X 0,Y 158.678,Z 357.934,A -85,B 0,C 180,E1 -25870.272,E2 -25870.272} C_VEL
LIN {X 0,Y 153.795,Z 347.372,A -85,B 0,C 180,E1 -25873.138,E2 -25873.138} C_VEL
LIN {X 0,Y 148.164,Z 337.062,A -85,B 0,C 180,E1 -25876.763,E2 -25876.763} C_VEL
LIN {X 0,Y 143.245,Z 329.029,A -85,B 0,C 180,E1 -25880.376,E2 -25880.376} C_VEL
LIN {X 0,Y 139.678,Z 323.951,A -85,B 0,C 180,E1 -25883.346,E2 -25883.346} C_VEL
LIN {X 0,Y 137.289,Z 320.515,A -85,B 0,C 180,E1 -25885.601,E2 -25885.601} C_VEL
LIN {X 0,Y 134.204,Z 316.243,A -85,B 0,C 180,E1 -25888.913,E2 -25888.913} C_VEL
LIN {X 0,Y 131.554,Z 313.245,A -85,B 0,C 180,E1 -25892.197,E2 -25892.197} C_VEL
LIN {X 0,Y 130.574,Z 311.394,A -85,B 0,C 180,E1 -25893.703,E2 -25893.703} C_VEL
LIN {X 0,Y 127.898,Z 309.128,A -85,B 0,C 180,E1 -25898.112,E2 -25898.112} C_VEL
LIN {X 0,Y 126.647,Z 306.239,A -85,B 0,C 180,E1 -25901.292,E2 -25901.292} C_VEL
LIN {X 0,Y 125.742,Z 305.691,A -85,B 0,C 180,E1 -25903.777,E2 -25903.777} C_VEL
LIN {X 0,Y 124.45,Z 304.793,A -85,B 0,C 180,E1 -25910.251,E2 -25910.251} C_VEL
LIN {X 0,Y 125.361,Z 304.997,A -85,B 0,C 180,E1 -25920.358,E2 -25920.358} C_VEL
LIN {X 0,Y 126.832,Z 305.998,A -85,B 0,C 180,E1 -25924.672,E2 -25924.672} C_VEL
LIN {X 0,Y 128.414,Z 309.298,A -85,B 0,C 180,E1 -25928.413,E2 -25928.413} C_VEL
LIN {X 0,Y 130.918,Z 311.681,A -85,B 0,C 180,E1 -25932.404,E2 -25932.404} C_VEL
LIN {X 0,Y 133.28,Z 315.347,A -85,B 0,C 180,E1 -25935.658,E2 -25935.658} C_VEL
LIN {X 0,Y 134.707,Z 316.872,A -85,B 0,C 180,E1 -25937.29,E2 -25937.29} C_VEL
LIN {X 0,Y 137.365,Z 320.656,A -85,B 0,C 180,E1 -25940.109,E2 -25940.109} C_VEL
LIN {X 0,Y 139.005,Z 323.047,A -85,B 0,C 180,E1 -25941.677,E2 -25941.677} C_VEL
LIN {X 0,Y 141.676,Z 326.779,A -85,B 0,C 180,E1 -25943.991,E2 -25943.991} C_VEL
LIN {X 0,Y 145.788,Z 333.183,A -85,B 0,C 180,E1 -25947.186,E2 -25947.186} C_VEL
LIN {X 0,Y 151.049,Z 342.301,A -85,B 0,C 180,E1 -25950.788,E2 -25950.788} C_VEL
LIN {X 0,Y 155.795,Z 354.612,A -85,B 0,C 180,E1 -25953.908,E2 -25953.908} C_VEL
LIN {X 0,Y 158.766,Z 363.786,A -85,B 0,C 180,E1 -25955.781,E2 -25955.781} C_VEL
LIN {X 0,Y 154.229,Z 421.794,A -85,B 0,C 180,E1 -25957.988,E2 -25957.988} C_VEL
LIN {X 0,Y 152.044,Z 435.996,A -85,B 0,C 180,E1 -25958.871,E2 -25958.871} C_VEL
LIN {X 0,Y 149.479,Z 447.803,A -85,B 0,C 180,E1 -25959.919,E2 -25959.919} C_VEL
LIN {X 0,Y 145.778,Z 461.426,A -85,B 0,C 180,E1 -25961.647,E2 -25961.647} C_VEL
LIN {X 0,Y 141.72,Z 473.452,A -85,B 0,C 180,E1 -25963.665,E2 -25963.665} C_VEL
LIN {X 0,Y 137.41,Z 485.162,A -85,B 0,C 180,E1 -25966.333,E2 -25966.333} C_VEL
LIN {X 0,Y 133.825,Z 493.069,A -85,B 0,C 180,E1 -25968.47,E2 -25968.47} C_VEL
LIN {X 0,Y 128.872,Z 503.663,A -85,B 0,C 180,E1 -25972.156,E2 -25972.156} C_VEL
LIN {X 0,Y 124.12,Z 513.207,A -85,B 0,C 180,E1 -25976.491,E2 -25976.491} C_VEL
LIN {X 0,Y 119.726,Z 521.933,A -85,B 0,C 180,E1 -25981.712,E2 -25981.712} C_VEL
LIN {X 0,Y 116.556,Z 528.654,A -85,B 0,C 180,E1 -25986.925,E2 -25986.925} C_VEL
LIN {X 0,Y 114.271,Z 533.879,A -85,B 0,C 180,E1 -25992.09,E2 -25992.09} C_VEL
LIN {X 0,Y 112.923,Z 538.101,A -85,B 0,C 180,E1 -25997.418,E2 -25997.418} C_VEL
LIN {X 0,Y 112.254,Z 541.433,A -85,B 0,C 180,E1 -26002.807,E2 -26002.807} C_VEL
LIN {X 0,Y 112.308,Z 544.517,A -85,B 0,C 180,E1 -26010,E2 -26010} C_VEL
LIN {X 0,Y 112.199,Z 545.508,A -85,B 0,C 180,E1 -26013.591,E2 -26013.591} C_VEL
LIN {X 0,Y 112.691,Z 546.483,A -85,B 0,C 180,E1 -26020.783,E2 -26020.783} C_VEL
LIN {X 0,Y 114.551,Z 546.157,A -85,B 0,C 180,E1 -26027.863,E2 -26027.863} C_VEL
LIN {X 0,Y 117.278,Z 544.931,A -85,B 0,C 180,E1 -26033.299,E2 -26033.299} C_VEL
LIN {X 0,Y 118.408,Z 544.065,A -85,B 0,C 180,E1 -26036.089,E2 -26036.089} C_VEL
LIN {X 0,Y 119.091,Z 542.272,A -85,B 0,C 180,E1 -26040.793,E2 -26040.793} C_VEL
LIN {X 0,Y 120.522,Z 539.888,A -85,B 0,C 180,E1 -26045.345,E2 -26045.345} C_VEL
LIN {X 0,Y 122.733,Z 538.083,A -85,B 0,C 180,E1 -26047.779,E2 -26047.779} C_VEL
LIN {X 0,Y 129.79,Z 533.173,A -85,B 0,C 180,E1 -26052.597,E2 -26052.597} C_VEL
LIN {X 0,Y 138.617,Z 526.101,A -85,B 0,C 180,E1 -26057.319,E2 -26057.319} C_VEL
LIN {X 0,Y 147.167,Z 518.329,A -85,B 0,C 180,E1 -26060.896,E2 -26060.896} C_VEL
LIN {X 0,Y 154.902,Z 510.165,A -85,B 0,C 180,E1 -26063.707,E2 -26063.707} C_VEL
LIN {X 0,Y 162.794,Z 500.569,A -85,B 0,C 180,E1 -26066.204,E2 -26066.204} C_VEL
LIN {X 0,Y 170.519,Z 489.823,A -85,B 0,C 180,E1 -26068.216,E2 -26068.216} C_VEL
LIN {X 0,Y 177.642,Z 477.969,A -85,B 0,C 180,E1 -26069.93,E2 -26069.93} C_VEL
LIN {X 0,Y 183.558,Z 466.305,A -85,B 0,C 180,E1 -26071.14,E2 -26071.14} C_VEL
LIN {X 0,Y 189.117,Z 452.624,A -85,B 0,C 180,E1 -26072.239,E2 -26072.239} C_VEL
LIN {X 0,Y 193.536,Z 438.305,A -85,B 0,C 180,E1 -26073.035,E2 -26073.035} C_VEL
LIN {X 0,Y 196.559,Z 424.495,A -85,B 0,C 180,E1 -26073.561,E2 -26073.561} C_VEL
LIN {X 0,Y 198.774,Z 406.84,A -85,B 0,C 180,E1 -26074.05,E2 -26074.05} C_VEL
LIN {X 0,Y 199.395,Z 400.408,A -85,B 0,C 180,E1 -26074.236,E2 -26074.236} C_VEL
LIN {X 0,Y 197.176,Z 393.67,A -85,B 0,C 180,E1 -26076.969,E2 -26076.969} C_VEL
LIN {X 0,Y 195.525,Z 389.207,A -85,B 0,C 180,E1 -26079.293,E2 -26079.293} C_VEL
LIN {X 0,Y 194.036,Z 385.329,A -85,B 0,C 180,E1 -26081.828,E2 -26081.828} C_VEL
LIN {X 0,Y 193.311,Z 383.634,A -85,B 0,C 180,E1 -26083.282,E2 -26083.282} C_VEL
LIN {X 0,Y 191.606,Z 379.933,A -85,B 0,C 180,E1 -26088.039,E2 -26088.039} C_VEL
LIN {X 0,Y 190.884,Z 379.082,A -85,B 0,C 180,E1 -26093.656,E2 -26093.656} C_VEL
LIN {X 0,Y 191.772,Z 379.714,A -85,B 0,C 180,E1 -26098.816,E2 -26098.816} C_VEL
LIN {X 0,Y 193.599,Z 383.947,A -85,B 0,C 180,E1 -26103.672,E2 -26103.672} C_VEL
LIN {X 0,Y 195.613,Z 388.208,A -85,B 0,C 180,E1 -26107.091,E2 -26107.091} C_VEL
LIN {X 0,Y 197.881,Z 392.916,A -85,B 0,C 180,E1 -26110.032,E2 -26110.032} C_VEL
LIN {X 0,Y 199.688,Z 396.953,A -85,B 0,C 180,E1 -26112.059,E2 -26112.059} C_VEL
LIN {X 0,Y 197.384,Z 417.692,A -85,B 0,C 180,E1 -26112.63,E2 -26112.63} C_VEL
LIN {X 0,Y 194.647,Z 431.557,A -85,B 0,C 180,E1 -26113.165,E2 -26113.165} C_VEL
LIN {X 0,Y 190.937,Z 444.654,A -85,B 0,C 180,E1 -26113.884,E2 -26113.884} C_VEL
LIN {X 0,Y 186.327,Z 457.261,A -85,B 0,C 180,E1 -26114.872,E2 -26114.872} C_VEL
LIN {X 0,Y 180.271,Z 470.423,A -85,B 0,C 180,E1 -26116.261,E2 -26116.261} C_VEL
LIN {X 0,Y 173.565,Z 482.304,A -85,B 0,C 180,E1 -26117.911,E2 -26117.911} C_VEL
LIN {X 0,Y 166.43,Z 492.972,A -85,B 0,C 180,E1 -26119.881,E2 -26119.881} C_VEL
LIN {X 0,Y 159.226,Z 502.13,A -85,B 0,C 180,E1 -26122.046,E2 -26122.046} C_VEL
LIN {X 0,Y 151.663,Z 510.506,A -85,B 0,C 180,E1 -26124.645,E2 -26124.645} C_VEL
LIN {X 0,Y 143.319,Z 518.58,A -85,B 0,C 180,E1 -26128.036,E2 -26128.036} C_VEL
LIN {X 0,Y 135.765,Z 524.937,A -85,B 0,C 180,E1 -26131.71,E2 -26131.71} C_VEL
LIN {X 0,Y 127.351,Z 531.126,A -85,B 0,C 180,E1 -26136.822,E2 -26136.822} C_VEL
LIN {X 0,Y 121.546,Z 534.763,A -85,B 0,C 180,E1 -26141.266,E2 -26141.266} C_VEL
LIN {X 0,Y 115.052,Z 538.235,A -85,B 0,C 180,E1 -26147.785,E2 -26147.785} C_VEL
LIN {X 0,Y 110.089,Z 540.192,A -85,B 0,C 180,E1 -26154.933,E2 -26154.933} C_VEL
LIN {X 0,Y 106.714,Z 540.688,A -85,B 0,C 180,E1 -26162.549,E2 -26162.549} C_VEL
